// Mitsubishi GX Works2 project: GCP-712ARB(2#)-20040003-220112   PLC: Q03UDV

PROGRAM 01INITI
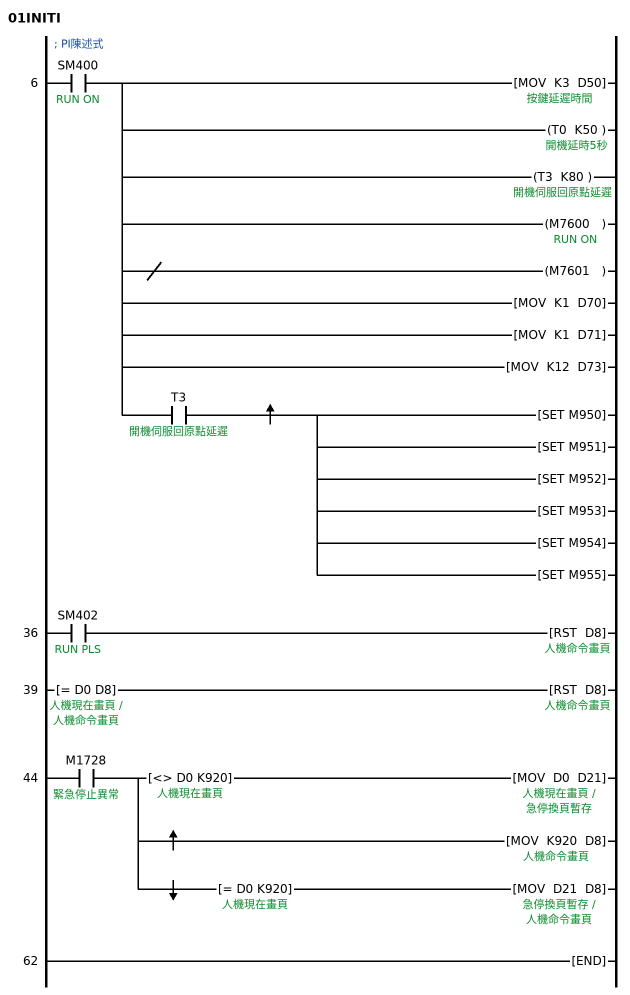
; PI陳述式
6     LD      SM400  ; RUN ON
      MOV     K3 D50  ; 按鍵延遲時間
      OUT     T0 K50  ; 開機延時5秒
      OUT     T3 K80  ; 開機伺服回原點延遲
      OUT     M7600  ; RUN ON
      MPS
      INV
      OUT     M7601
      MPP
      MOV     K1 D70
      MOV     K1 D71
      MOV     K12 D73
      AND     T3  ; 開機伺服回原點延遲
      MEP
      SET     M950
      SET     M951
      SET     M952
      SET     M953
      SET     M954
      SET     M955
36    LD      SM402  ; RUN PLS
      RST     D8  ; 人機命令畫頁
39    LD=     D0 D8  ; 人機現在畫頁 / 人機命令畫頁
      RST     D8  ; 人機命令畫頁
44    LD      M1728  ; 緊急停止異常
      MPS
      AND<>   D0 K920  ; 人機現在畫頁
      MOV     D0 D21  ; 急停換頁暫存
      MRD
      MEP
      MOV     K920 D8
      MPP
      MEF
      AND=    D0 K920  ; 人機現在畫頁
      MOV     D21 D8
62    END
END_PROGRAM

PROGRAM 02FUNC
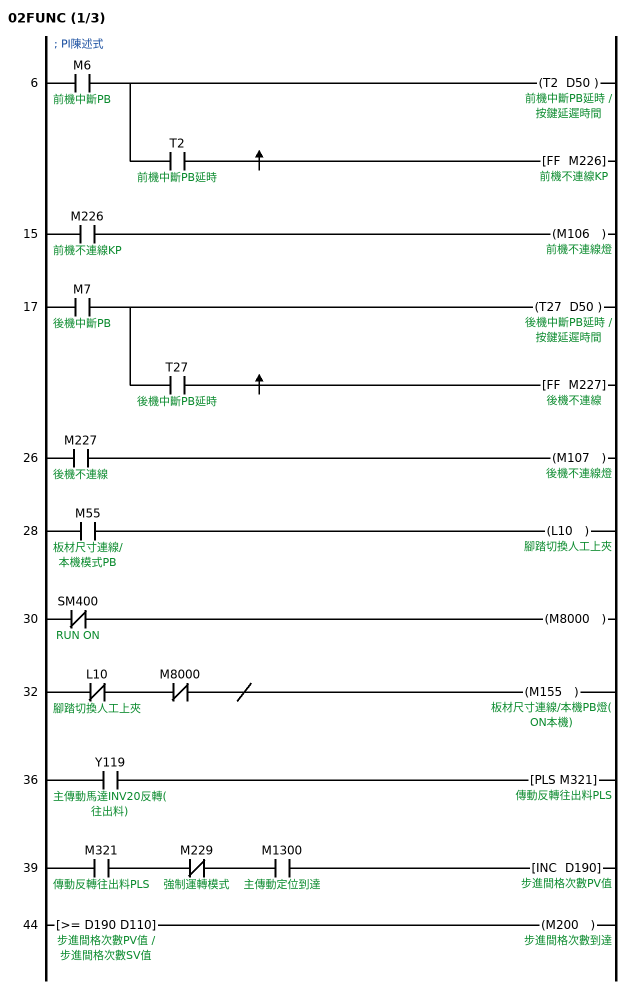
; PI陳述式
6     LD      M6  ; 前機中斷PB
      OUT     T2 D50  ; 前機中斷PB延時 / 按鍵延遲時間
      AND     T2  ; 前機中斷PB延時
      MEP
      FF      M226  ; 前機不連線KP
15    LD      M226  ; 前機不連線KP
      OUT     M106  ; 前機不連線燈
17    LD      M7  ; 後機中斷PB
      OUT     T27 D50  ; 後機中斷PB延時 / 按鍵延遲時間
      AND     T27  ; 後機中斷PB延時
      MEP
      FF      M227  ; 後機不連線
26    LD      M227  ; 後機不連線
      OUT     M107  ; 後機不連線燈
28    LD      M55  ; 板材尺寸連線/本機模式PB
      OUT     L10  ; 腳踏切換人工上夾
30    LDI     SM400  ; RUN ON
      OUT     M8000
32    LDI     L10  ; 腳踏切換人工上夾
      ANI     M8000
      INV
      OUT     M155  ; 板材尺寸連線/本機PB燈(ON本機)
36    LD      Y119  ; 主傳動馬達INV20反轉(往出料)
      PLS     M321  ; 傳動反轉往出料PLS
39    LD      M321  ; 傳動反轉往出料PLS
      ANI     M229  ; 強制運轉模式
      AND     M1300  ; 主傳動定位到達
      INC     D190  ; 步進間格次數PV值
44    LD>=    D190 D110  ; 步進間格次數PV值 / 步進間格次數SV值
      OUT     M200  ; 步進間格次數到達
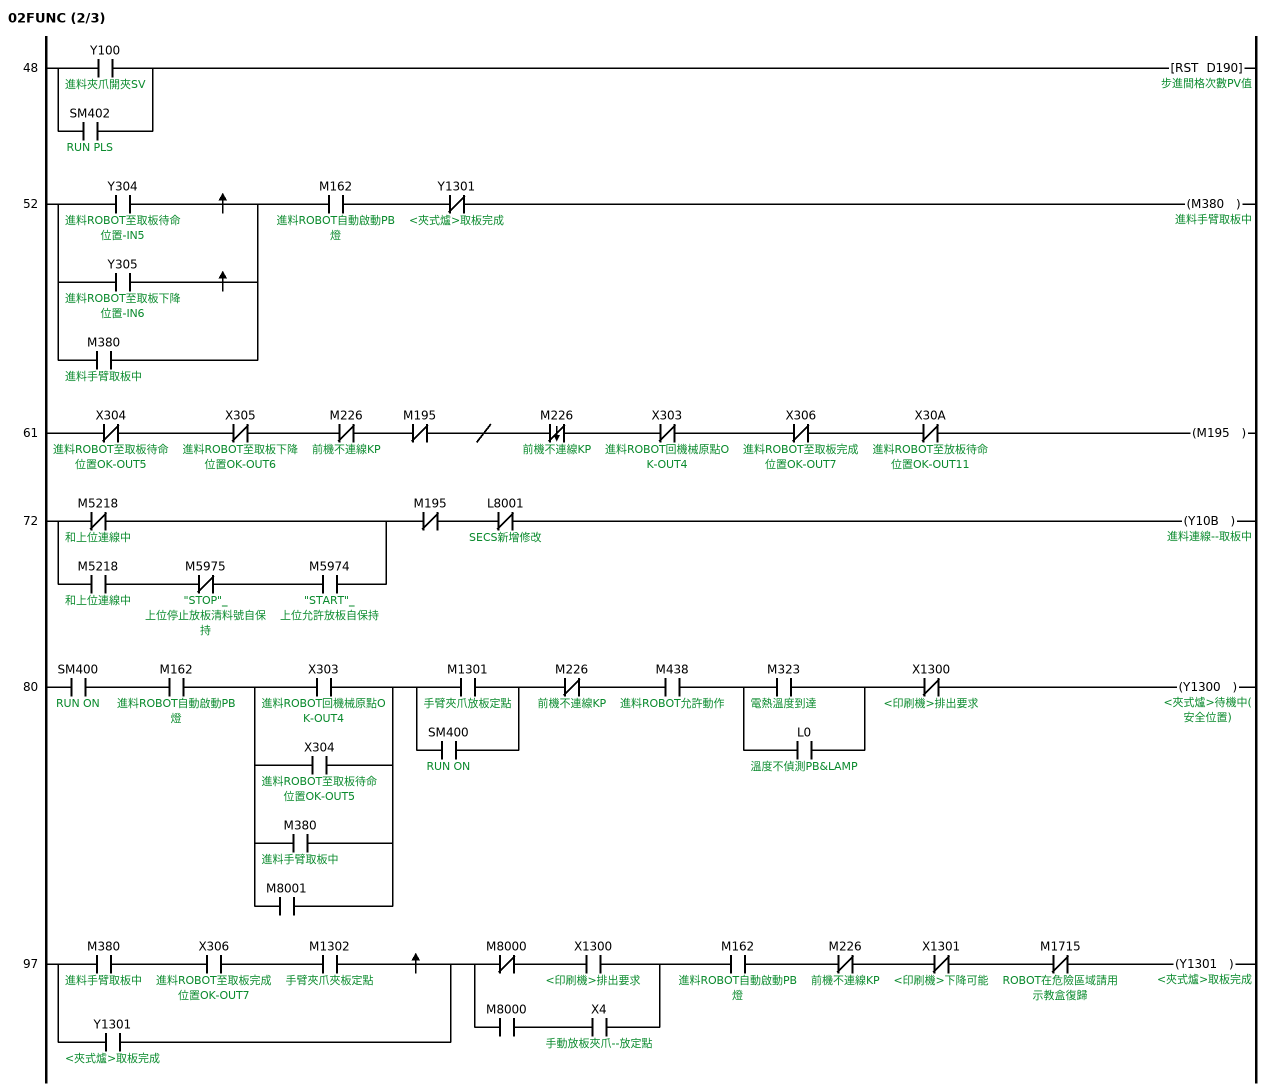
48    LD      Y100  ; 進料夾爪開夾SV
      OR      SM402  ; RUN PLS
      RST     D190  ; 步進間格次數PV值
52    LD      Y304  ; 進料ROBOT至取板待命位置-IN5
      MEP
      LD      Y305  ; 進料ROBOT至取板下降位置-IN6
      MEP
      ORB
      OR      M380  ; 進料手臂取板中
      AND     M162  ; 進料ROBOT自動啟動PB燈
      ANI     Y1301  ; <夾式爐>取板完成
      OUT     M380  ; 進料手臂取板中
61    LDI     X304  ; 進料ROBOT至取板待命位置OK-OUT5
      ANI     X305  ; 進料ROBOT至取板下降位置OK-OUT6
      ANI     M226  ; 前機不連線KP
      ANI     M195
      INV
      ANDFI   M226  ; 前機不連線KP
      ANI     X303  ; 進料ROBOT回機械原點OK-OUT4
      ANI     X306  ; 進料ROBOT至取板完成位置OK-OUT7
      ANI     X30A  ; 進料ROBOT至放板待命位置OK-OUT11
      OUT     M195
72    LDI     M5218  ; 和上位連線中
      LD      M5218  ; 和上位連線中
      ANI     M5975  ; "STOP"_ 上位停止放板清料號自保持
      AND     M5974  ; "START"_上位允許放板自保持
      ORB
      ANI     M195
      ANI     L8001  ; SECS新增修改
      OUT     Y10B  ; 進料連線--取板中
80    LD      SM400  ; RUN ON
      AND     M162  ; 進料ROBOT自動啟動PB燈
      LD      X303  ; 進料ROBOT回機械原點OK-OUT4
      OR      X304  ; 進料ROBOT至取板待命位置OK-OUT5
      OR      M380  ; 進料手臂取板中
      OR      M8001
      ANB
      LD      M1301  ; 手臂夾爪放板定點
      OR      SM400  ; RUN ON
      ANB
      ANI     M226  ; 前機不連線KP
      AND     M438  ; 進料ROBOT允許動作
      LD      M323  ; 電熱溫度到達
      OR      L0  ; 溫度不偵測PB&LAMP
      ANB
      ANI     X1300  ; <印刷機>排出要求
      OUT     Y1300  ; <夾式爐>待機中(安全位置)
97    LD      M380  ; 進料手臂取板中
      AND     X306  ; 進料ROBOT至取板完成位置OK-OUT7
      AND     M1302  ; 手臂夾爪夾板定點
      MEP
      OR      Y1301  ; <夾式爐>取板完成
      LDI     M8000
      AND     X1300  ; <印刷機>排出要求
      LD      M8000
      AND     X4  ; 手動放板夾爪--放定點
      ORB
      ANB
      AND     M162  ; 進料ROBOT自動啟動PB燈
      ANI     M226  ; 前機不連線KP
      ANI     X1301  ; <印刷機>下降可能
      ANI     M1715  ; ROBOT在危險區域請用示教盒復歸
      OUT     Y1301  ; <夾式爐>取板完成
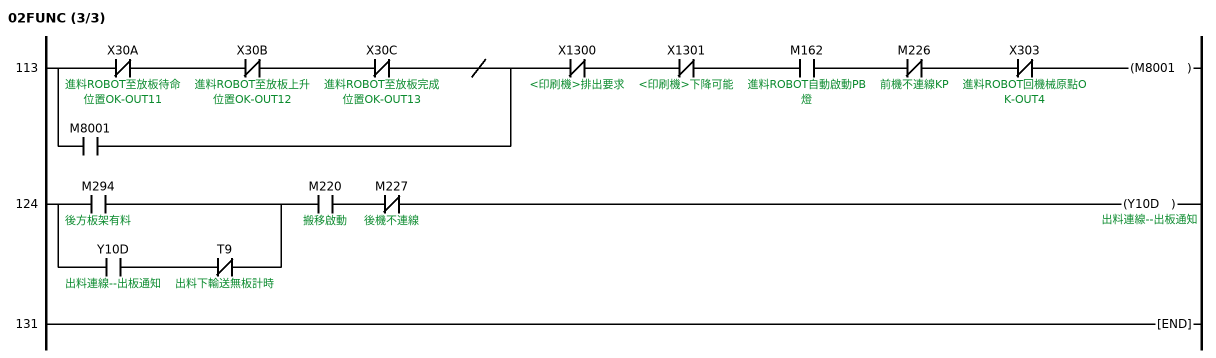
113   LDI     X30A  ; 進料ROBOT至放板待命位置OK-OUT11
      ANI     X30B  ; 進料ROBOT至放板上升位置OK-OUT12
      ANI     X30C  ; 進料ROBOT至放板完成位置OK-OUT13
      INV
      OR      M8001
      ANI     X1300  ; <印刷機>排出要求
      ANI     X1301  ; <印刷機>下降可能
      AND     M162  ; 進料ROBOT自動啟動PB燈
      ANI     M226  ; 前機不連線KP
      ANI     X303  ; 進料ROBOT回機械原點OK-OUT4
      OUT     M8001
124   LD      M294  ; 後方板架有料
      LD      Y10D  ; 出料連線--出板通知
      ANI     T9  ; 出料下輸送無板計時
      ORB
      AND     M220  ; 搬移啟動
      ANI     M227  ; 後機不連線
      OUT     Y10D  ; 出料連線--出板通知
131   END
END_PROGRAM

PROGRAM 03ORIGIN
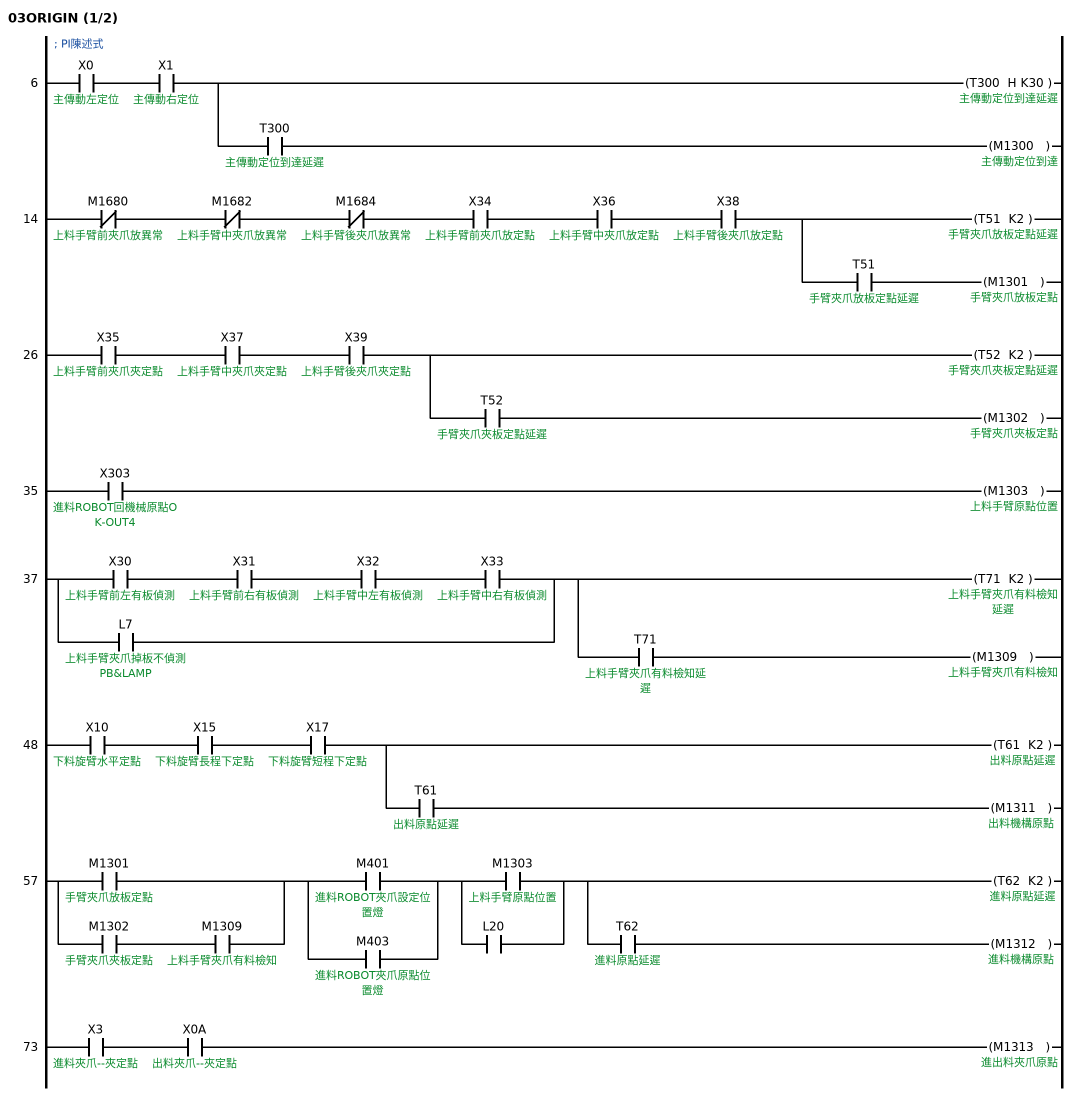
; PI陳述式
6     LD      X0  ; 主傳動左定位
      AND     X1  ; 主傳動右定位
      OUTH    T300 K30  ; 主傳動定位到達延遲
      AND     T300  ; 主傳動定位到達延遲
      OUT     M1300  ; 主傳動定位到達
14    LDI     M1680  ; 上料手臂前夾爪放異常
      ANI     M1682  ; 上料手臂中夾爪放異常
      ANI     M1684  ; 上料手臂後夾爪放異常
      AND     X34  ; 上料手臂前夾爪放定點
      AND     X36  ; 上料手臂中夾爪放定點
      AND     X38  ; 上料手臂後夾爪放定點
      OUT     T51 K2  ; 手臂夾爪放板定點延遲
      AND     T51  ; 手臂夾爪放板定點延遲
      OUT     M1301  ; 手臂夾爪放板定點
26    LD      X35  ; 上料手臂前夾爪夾定點
      AND     X37  ; 上料手臂中夾爪夾定點
      AND     X39  ; 上料手臂後夾爪夾定點
      OUT     T52 K2  ; 手臂夾爪夾板定點延遲
      AND     T52  ; 手臂夾爪夾板定點延遲
      OUT     M1302  ; 手臂夾爪夾板定點
35    LD      X303  ; 進料ROBOT回機械原點OK-OUT4
      OUT     M1303  ; 上料手臂原點位置
37    LD      X30  ; 上料手臂前左有板偵測
      AND     X31  ; 上料手臂前右有板偵測
      AND     X32  ; 上料手臂中左有板偵測
      AND     X33  ; 上料手臂中右有板偵測
      OR      L7  ; 上料手臂夾爪掉板不偵測PB&LAMP
      OUT     T71 K2  ; 上料手臂夾爪有料檢知延遲
      AND     T71  ; 上料手臂夾爪有料檢知延遲
      OUT     M1309  ; 上料手臂夾爪有料檢知
48    LD      X10  ; 下料旋臂水平定點
      AND     X15  ; 下料旋臂長程下定點
      AND     X17  ; 下料旋臂短程下定點
      OUT     T61 K2  ; 出料原點延遲
      AND     T61  ; 出料原點延遲
      OUT     M1311  ; 出料機構原點
57    LD      M1301  ; 手臂夾爪放板定點
      LD      M1302  ; 手臂夾爪夾板定點
      AND     M1309  ; 上料手臂夾爪有料檢知
      ORB
      LD      M401  ; 進料ROBOT夾爪設定位置燈
      OR      M403  ; 進料ROBOT夾爪原點位置燈
      ANB
      LD      M1303  ; 上料手臂原點位置
      OR      L20
      ANB
      OUT     T62 K2  ; 進料原點延遲
      AND     T62  ; 進料原點延遲
      OUT     M1312  ; 進料機構原點
73    LD      X3  ; 進料夾爪--夾定點
      AND     X0A  ; 出料夾爪--夾定點
      OUT     M1313  ; 進出料夾爪原點
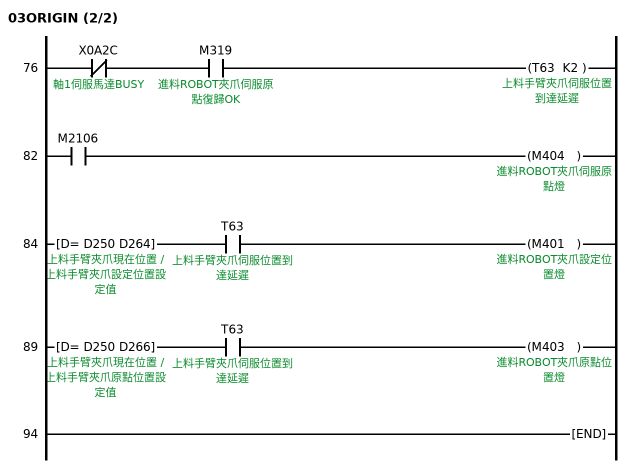
76    LDI     X0A2C  ; 軸1伺服馬達BUSY
      AND     M319  ; 進料ROBOT夾爪伺服原點復歸OK
      OUT     T63 K2  ; 上料手臂夾爪伺服位置到達延遲
82    LD      M2106
      OUT     M404  ; 進料ROBOT夾爪伺服原點燈
84    LDD=    D250 D264  ; 上料手臂夾爪現在位置 / 上料手臂夾爪設定位置設定值
      AND     T63  ; 上料手臂夾爪伺服位置到達延遲
      OUT     M401  ; 進料ROBOT夾爪設定位置燈
89    LDD=    D250 D266  ; 上料手臂夾爪現在位置 / 上料手臂夾爪原點位置設定值
      AND     T63  ; 上料手臂夾爪伺服位置到達延遲
      OUT     M403  ; 進料ROBOT夾爪原點位置燈
94    END
END_PROGRAM

PROGRAM 04LOAD
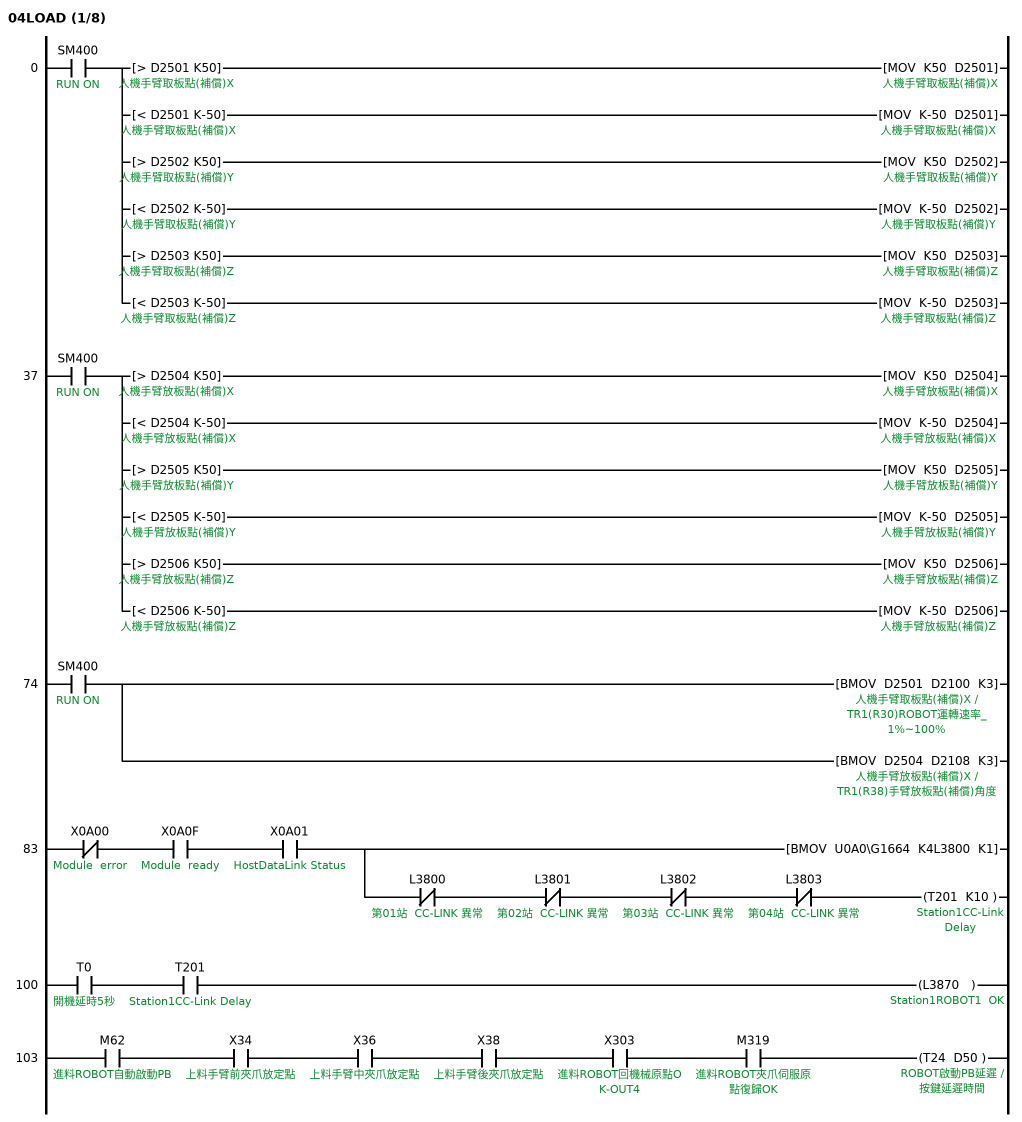
0     LD      SM400  ; RUN ON
      MPS
      AND>    D2501 K50  ; 人機手臂取板點(補償)X
      MOV     K50 D2501
      MRD
      AND<    D2501 K-50  ; 人機手臂取板點(補償)X
      MOV     K-50 D2501
      MRD
      AND>    D2502 K50  ; 人機手臂取板點(補償)Y
      MOV     K50 D2502
      MRD
      AND<    D2502 K-50  ; 人機手臂取板點(補償)Y
      MOV     K-50 D2502
      MRD
      AND>    D2503 K50  ; 人機手臂取板點(補償)Z
      MOV     K50 D2503
      MPP
      AND<    D2503 K-50  ; 人機手臂取板點(補償)Z
      MOV     K-50 D2503
37    LD      SM400  ; RUN ON
      MPS
      AND>    D2504 K50  ; 人機手臂放板點(補償)X
      MOV     K50 D2504
      MRD
      AND<    D2504 K-50  ; 人機手臂放板點(補償)X
      MOV     K-50 D2504
      MRD
      AND>    D2505 K50  ; 人機手臂放板點(補償)Y
      MOV     K50 D2505
      MRD
      AND<    D2505 K-50  ; 人機手臂放板點(補償)Y
      MOV     K-50 D2505
      MRD
      AND>    D2506 K50  ; 人機手臂放板點(補償)Z
      MOV     K50 D2506
      MPP
      AND<    D2506 K-50  ; 人機手臂放板點(補償)Z
      MOV     K-50 D2506
74    LD      SM400  ; RUN ON
      BMOV    D2501 D2100 K3  ; TR1(R30)ROBOT運轉速率_1%~100%
      BMOV    D2504 D2108 K3  ; TR1(R38)手臂放板點(補償)角度
83    LDI     X0A00  ; Module  error
      AND     X0A0F  ; Module  ready
      AND     X0A01  ; HostDataLink Status
      BMOV    U0A0\G1664 K4L3800 K1  ; 第01站  CC-LINK 異常
      ANI     L3800  ; 第01站  CC-LINK 異常
      ANI     L3801  ; 第02站  CC-LINK 異常
      ANI     L3802  ; 第03站  CC-LINK 異常
      ANI     L3803  ; 第04站  CC-LINK 異常
      OUT     T201 K10  ; Station1CC-Link Delay
100   LD      T0  ; 開機延時5秒
      AND     T201  ; Station1CC-Link Delay
      OUT     L3870  ; Station1ROBOT1  OK
103   LD      M62  ; 進料ROBOT自動啟動PB
      AND     X34  ; 上料手臂前夾爪放定點
      AND     X36  ; 上料手臂中夾爪放定點
      AND     X38  ; 上料手臂後夾爪放定點
      AND     X303  ; 進料ROBOT回機械原點OK-OUT4
      AND     M319  ; 進料ROBOT夾爪伺服原點復歸OK
      OUT     T24 D50  ; ROBOT啟動PB延遲 / 按鍵延遲時間
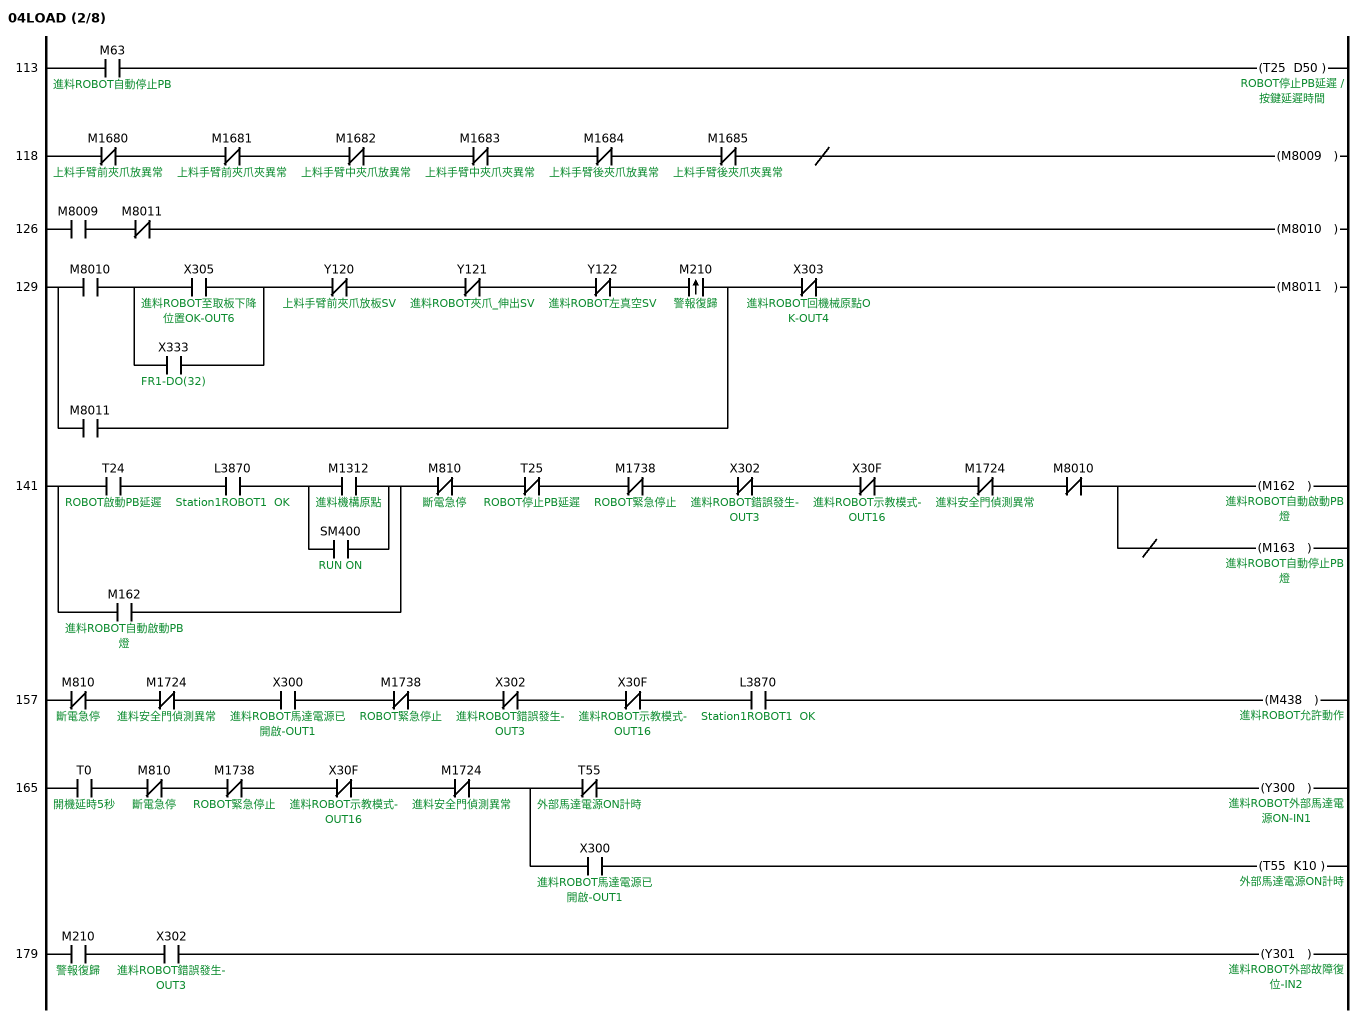
113   LD      M63  ; 進料ROBOT自動停止PB
      OUT     T25 D50  ; ROBOT停止PB延遲 / 按鍵延遲時間
118   LDI     M1680  ; 上料手臂前夾爪放異常
      ANI     M1681  ; 上料手臂前夾爪夾異常
      ANI     M1682  ; 上料手臂中夾爪放異常
      ANI     M1683  ; 上料手臂中夾爪夾異常
      ANI     M1684  ; 上料手臂後夾爪放異常
      ANI     M1685  ; 上料手臂後夾爪夾異常
      INV
      OUT     M8009
126   LD      M8009
      ANI     M8011
      OUT     M8010
129   LD      M8010
      LD      X305  ; 進料ROBOT至取板下降位置OK-OUT6
      OR      X333  ; FR1-DO(32)
      ANB
      ANI     Y120  ; 上料手臂前夾爪放板SV
      ANI     Y121  ; 進料ROBOT夾爪_伸出SV
      ANI     Y122  ; 進料ROBOT左真空SV
      ANDP    M210  ; 警報復歸
      OR      M8011
      ANI     X303  ; 進料ROBOT回機械原點OK-OUT4
      OUT     M8011
141   LD      T24  ; ROBOT啟動PB延遲
      AND     L3870  ; Station1ROBOT1  OK
      LD      M1312  ; 進料機構原點
      OR      SM400  ; RUN ON
      ANB
      OR      M162  ; 進料ROBOT自動啟動PB燈
      ANI     M810  ; 斷電急停
      ANI     T25  ; ROBOT停止PB延遲
      ANI     M1738  ; ROBOT緊急停止
      ANI     X302  ; 進料ROBOT錯誤發生-OUT3
      ANI     X30F  ; 進料ROBOT示教模式-OUT16
      ANI     M1724  ; 進料安全門偵測異常
      ANI     M8010
      OUT     M162  ; 進料ROBOT自動啟動PB燈
      INV
      OUT     M163  ; 進料ROBOT自動停止PB燈
157   LDI     M810  ; 斷電急停
      ANI     M1724  ; 進料安全門偵測異常
      AND     X300  ; 進料ROBOT馬達電源已開啟-OUT1
      ANI     M1738  ; ROBOT緊急停止
      ANI     X302  ; 進料ROBOT錯誤發生-OUT3
      ANI     X30F  ; 進料ROBOT示教模式-OUT16
      AND     L3870  ; Station1ROBOT1  OK
      OUT     M438  ; 進料ROBOT允許動作
165   LD      T0  ; 開機延時5秒
      ANI     M810  ; 斷電急停
      ANI     M1738  ; ROBOT緊急停止
      ANI     X30F  ; 進料ROBOT示教模式-OUT16
      ANI     M1724  ; 進料安全門偵測異常
      MPS
      ANI     T55  ; 外部馬達電源ON計時
      OUT     Y300  ; 進料ROBOT外部馬達電源ON-IN1
      MPP
      AND     X300  ; 進料ROBOT馬達電源已開啟-OUT1
      OUT     T55 K10  ; 外部馬達電源ON計時
179   LD      M210  ; 警報復歸
      AND     X302  ; 進料ROBOT錯誤發生-OUT3
      OUT     Y301  ; 進料ROBOT外部故障復位-IN2
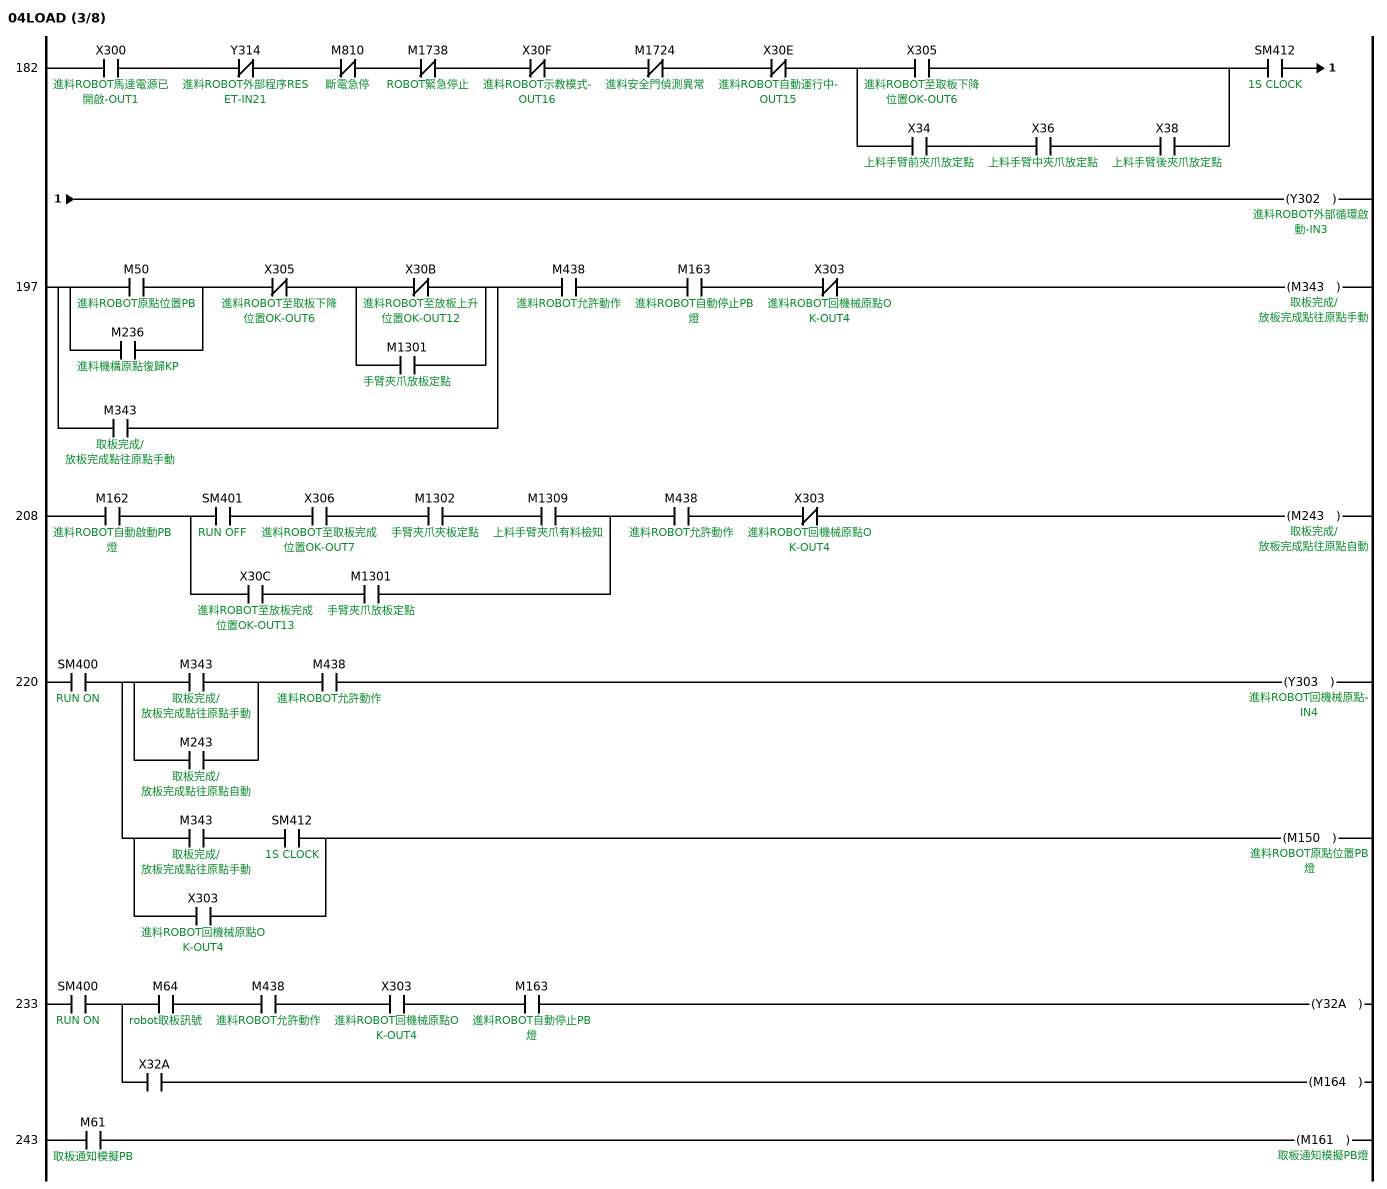
182   LD      X300  ; 進料ROBOT馬達電源已開啟-OUT1
      ANI     Y314  ; 進料ROBOT外部程序RESET-IN21
      ANI     M810  ; 斷電急停
      ANI     M1738  ; ROBOT緊急停止
      ANI     X30F  ; 進料ROBOT示教模式-OUT16
      ANI     M1724  ; 進料安全門偵測異常
      ANI     X30E  ; 進料ROBOT自動運行中-OUT15
      LD      X305  ; 進料ROBOT至取板下降位置OK-OUT6
      LD      X34  ; 上料手臂前夾爪放定點
      AND     X36  ; 上料手臂中夾爪放定點
      AND     X38  ; 上料手臂後夾爪放定點
      ORB
      ANB
      AND     SM412  ; 1S CLOCK
      OUT     Y302  ; 進料ROBOT外部循環啟動-IN3
197   LD      M50  ; 進料ROBOT原點位置PB
      OR      M236  ; 進料機構原點復歸KP
      ANI     X305  ; 進料ROBOT至取板下降位置OK-OUT6
      LDI     X30B  ; 進料ROBOT至放板上升位置OK-OUT12
      OR      M1301  ; 手臂夾爪放板定點
      ANB
      OR      M343  ; 取板完成/放板完成點往原點手動
      AND     M438  ; 進料ROBOT允許動作
      AND     M163  ; 進料ROBOT自動停止PB燈
      ANI     X303  ; 進料ROBOT回機械原點OK-OUT4
      OUT     M343  ; 取板完成/放板完成點往原點手動
208   LD      M162  ; 進料ROBOT自動啟動PB燈
      LD      SM401  ; RUN OFF
      AND     X306  ; 進料ROBOT至取板完成位置OK-OUT7
      AND     M1302  ; 手臂夾爪夾板定點
      AND     M1309  ; 上料手臂夾爪有料檢知
      LD      X30C  ; 進料ROBOT至放板完成位置OK-OUT13
      AND     M1301  ; 手臂夾爪放板定點
      ORB
      ANB
      AND     M438  ; 進料ROBOT允許動作
      ANI     X303  ; 進料ROBOT回機械原點OK-OUT4
      OUT     M243  ; 取板完成/放板完成點往原點自動
220   LD      SM400  ; RUN ON
      MPS
      LD      M343  ; 取板完成/放板完成點往原點手動
      OR      M243  ; 取板完成/放板完成點往原點自動
      ANB
      AND     M438  ; 進料ROBOT允許動作
      OUT     Y303  ; 進料ROBOT回機械原點-IN4
      MPP
      LD      M343  ; 取板完成/放板完成點往原點手動
      AND     SM412  ; 1S CLOCK
      OR      X303  ; 進料ROBOT回機械原點OK-OUT4
      ANB
      OUT     M150  ; 進料ROBOT原點位置PB燈
233   LD      SM400  ; RUN ON
      MPS
      AND     M64  ; robot取板訊號
      AND     M438  ; 進料ROBOT允許動作
      AND     X303  ; 進料ROBOT回機械原點OK-OUT4
      AND     M163  ; 進料ROBOT自動停止PB燈
      OUT     Y32A
      MPP
      AND     X32A
      OUT     M164
243   LD      M61  ; 取板通知模擬PB
      OUT     M161  ; 取板通知模擬PB燈
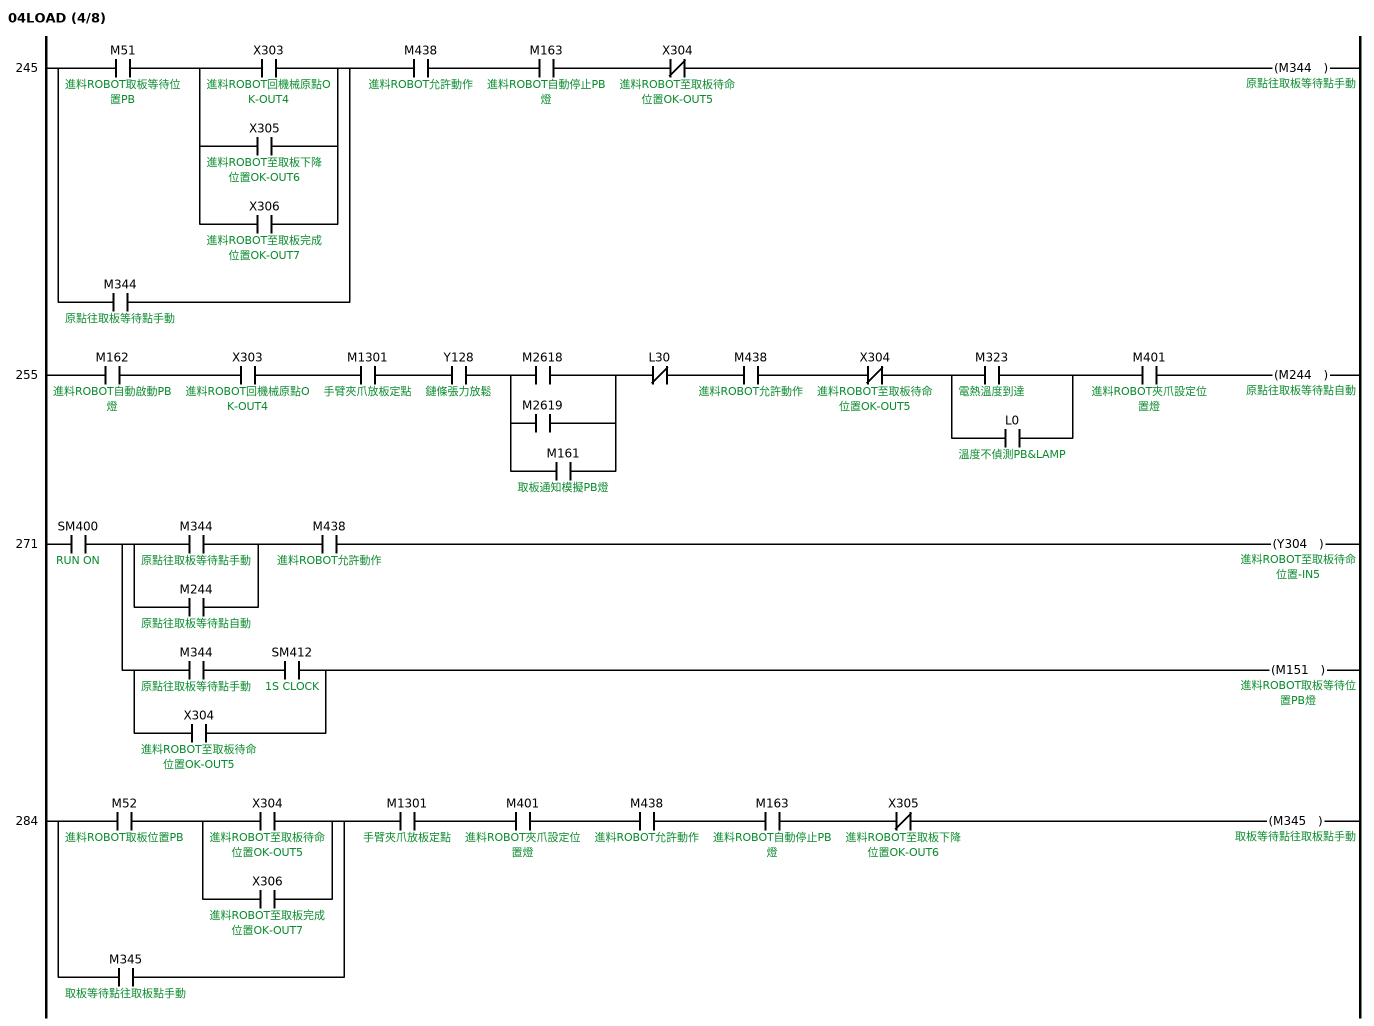
245   LD      M51  ; 進料ROBOT取板等待位置PB
      LD      X303  ; 進料ROBOT回機械原點OK-OUT4
      OR      X305  ; 進料ROBOT至取板下降位置OK-OUT6
      OR      X306  ; 進料ROBOT至取板完成位置OK-OUT7
      ANB
      OR      M344  ; 原點往取板等待點手動
      AND     M438  ; 進料ROBOT允許動作
      AND     M163  ; 進料ROBOT自動停止PB燈
      ANI     X304  ; 進料ROBOT至取板待命位置OK-OUT5
      OUT     M344  ; 原點往取板等待點手動
255   LD      M162  ; 進料ROBOT自動啟動PB燈
      AND     X303  ; 進料ROBOT回機械原點OK-OUT4
      AND     M1301  ; 手臂夾爪放板定點
      AND     Y128  ; 鏈條張力放鬆
      LD      M2618
      OR      M2619
      OR      M161  ; 取板通知模擬PB燈
      ANB
      ANI     L30
      AND     M438  ; 進料ROBOT允許動作
      ANI     X304  ; 進料ROBOT至取板待命位置OK-OUT5
      LD      M323  ; 電熱溫度到達
      OR      L0  ; 溫度不偵測PB&LAMP
      ANB
      AND     M401  ; 進料ROBOT夾爪設定位置燈
      OUT     M244  ; 原點往取板等待點自動
271   LD      SM400  ; RUN ON
      MPS
      LD      M344  ; 原點往取板等待點手動
      OR      M244  ; 原點往取板等待點自動
      ANB
      AND     M438  ; 進料ROBOT允許動作
      OUT     Y304  ; 進料ROBOT至取板待命位置-IN5
      MPP
      LD      M344  ; 原點往取板等待點手動
      AND     SM412  ; 1S CLOCK
      OR      X304  ; 進料ROBOT至取板待命位置OK-OUT5
      ANB
      OUT     M151  ; 進料ROBOT取板等待位置PB燈
284   LD      M52  ; 進料ROBOT取板位置PB
      LD      X304  ; 進料ROBOT至取板待命位置OK-OUT5
      OR      X306  ; 進料ROBOT至取板完成位置OK-OUT7
      ANB
      OR      M345  ; 取板等待點往取板點手動
      AND     M1301  ; 手臂夾爪放板定點
      AND     M401  ; 進料ROBOT夾爪設定位置燈
      AND     M438  ; 進料ROBOT允許動作
      AND     M163  ; 進料ROBOT自動停止PB燈
      ANI     X305  ; 進料ROBOT至取板下降位置OK-OUT6
      OUT     M345  ; 取板等待點往取板點手動
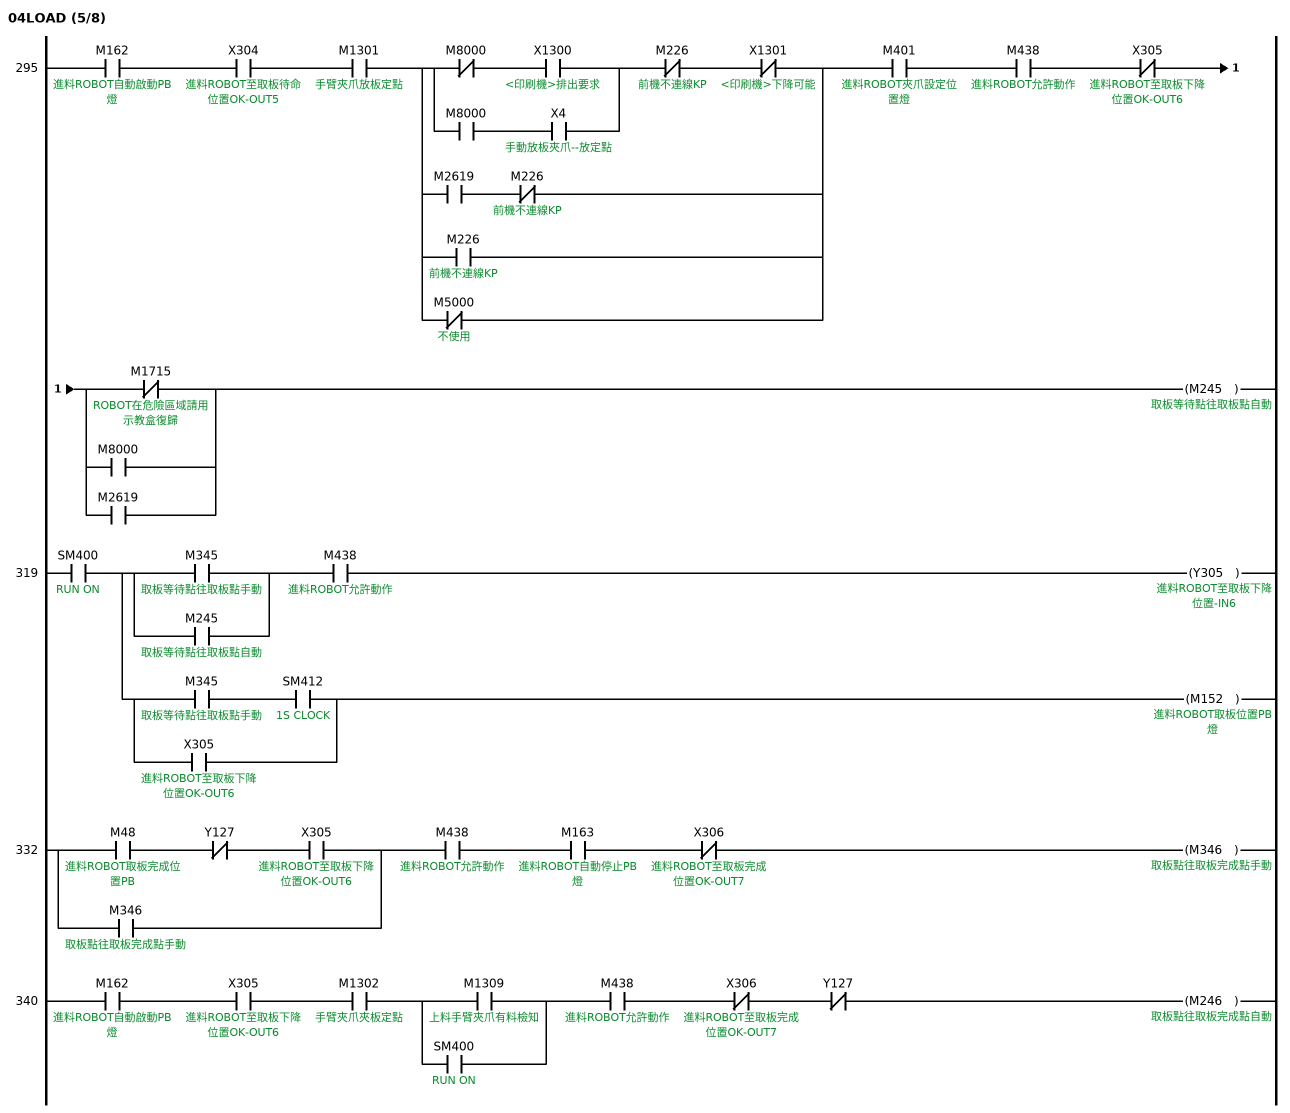
295   LD      M162  ; 進料ROBOT自動啟動PB燈
      AND     X304  ; 進料ROBOT至取板待命位置OK-OUT5
      AND     M1301  ; 手臂夾爪放板定點
      LDI     M8000
      AND     X1300  ; <印刷機>排出要求
      LD      M8000
      AND     X4  ; 手動放板夾爪--放定點
      ORB
      ANI     M226  ; 前機不連線KP
      ANI     X1301  ; <印刷機>下降可能
      LD      M2619
      ANI     M226  ; 前機不連線KP
      ORB
      OR      M226  ; 前機不連線KP
      ORI     M5000  ; 不使用
      ANB
      AND     M401  ; 進料ROBOT夾爪設定位置燈
      AND     M438  ; 進料ROBOT允許動作
      ANI     X305  ; 進料ROBOT至取板下降位置OK-OUT6
      LDI     M1715  ; ROBOT在危險區域請用示教盒復歸
      OR      M8000
      OR      M2619
      ANB
      OUT     M245  ; 取板等待點往取板點自動
319   LD      SM400  ; RUN ON
      MPS
      LD      M345  ; 取板等待點往取板點手動
      OR      M245  ; 取板等待點往取板點自動
      ANB
      AND     M438  ; 進料ROBOT允許動作
      OUT     Y305  ; 進料ROBOT至取板下降位置-IN6
      MPP
      LD      M345  ; 取板等待點往取板點手動
      AND     SM412  ; 1S CLOCK
      OR      X305  ; 進料ROBOT至取板下降位置OK-OUT6
      ANB
      OUT     M152  ; 進料ROBOT取板位置PB燈
332   LD      M48  ; 進料ROBOT取板完成位置PB
      ANI     Y127
      AND     X305  ; 進料ROBOT至取板下降位置OK-OUT6
      OR      M346  ; 取板點往取板完成點手動
      AND     M438  ; 進料ROBOT允許動作
      AND     M163  ; 進料ROBOT自動停止PB燈
      ANI     X306  ; 進料ROBOT至取板完成位置OK-OUT7
      OUT     M346  ; 取板點往取板完成點手動
340   LD      M162  ; 進料ROBOT自動啟動PB燈
      AND     X305  ; 進料ROBOT至取板下降位置OK-OUT6
      AND     M1302  ; 手臂夾爪夾板定點
      LD      M1309  ; 上料手臂夾爪有料檢知
      OR      SM400  ; RUN ON
      ANB
      AND     M438  ; 進料ROBOT允許動作
      ANI     X306  ; 進料ROBOT至取板完成位置OK-OUT7
      ANI     Y127
      OUT     M246  ; 取板點往取板完成點自動
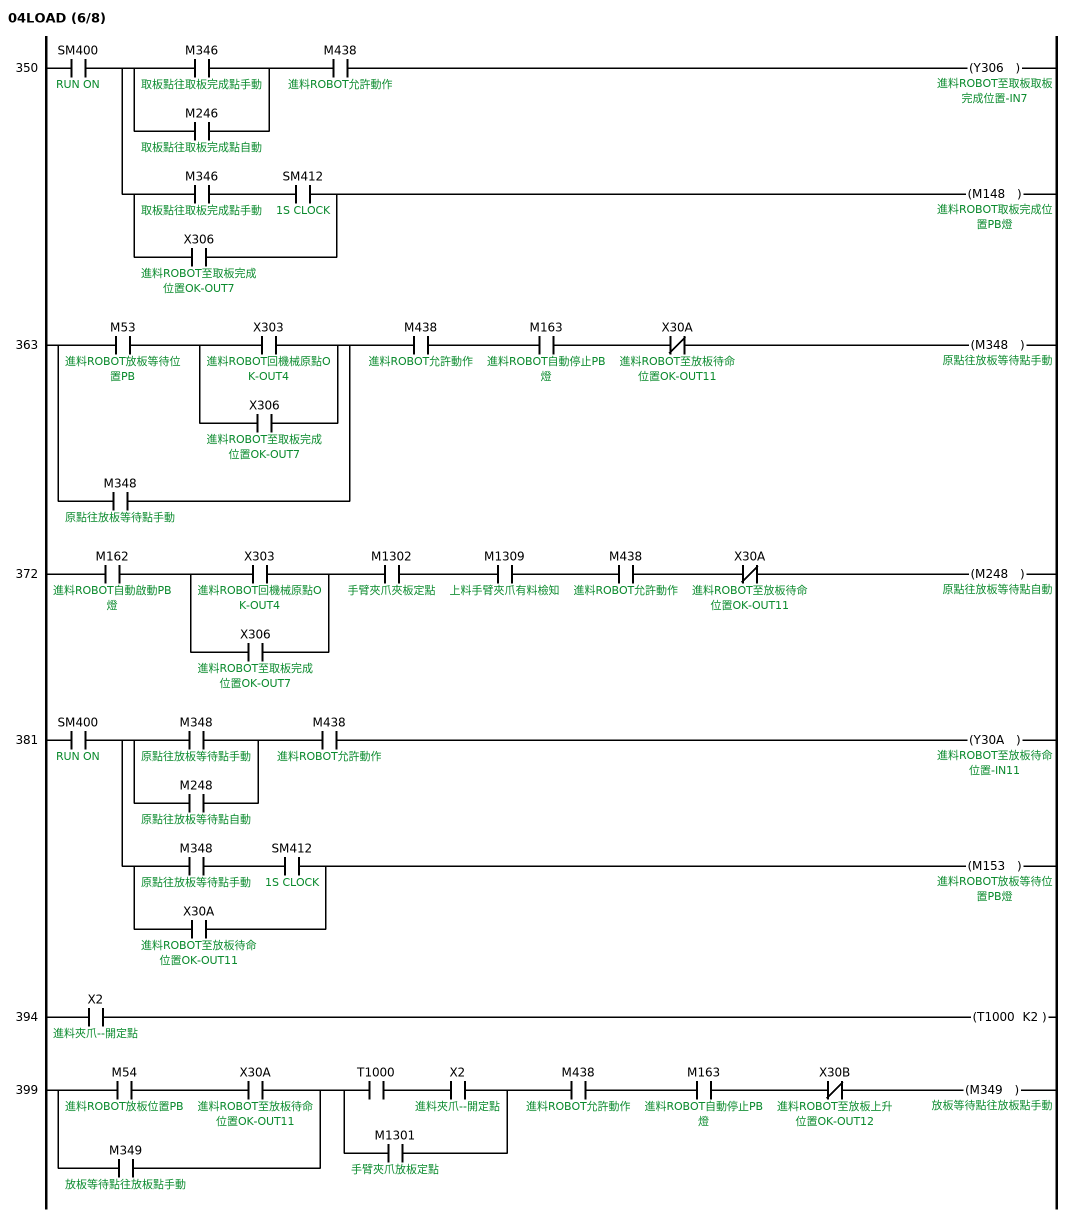
350   LD      SM400  ; RUN ON
      MPS
      LD      M346  ; 取板點往取板完成點手動
      OR      M246  ; 取板點往取板完成點自動
      ANB
      AND     M438  ; 進料ROBOT允許動作
      OUT     Y306  ; 進料ROBOT至取板取板完成位置-IN7
      MPP
      LD      M346  ; 取板點往取板完成點手動
      AND     SM412  ; 1S CLOCK
      OR      X306  ; 進料ROBOT至取板完成位置OK-OUT7
      ANB
      OUT     M148  ; 進料ROBOT取板完成位置PB燈
363   LD      M53  ; 進料ROBOT放板等待位置PB
      LD      X303  ; 進料ROBOT回機械原點OK-OUT4
      OR      X306  ; 進料ROBOT至取板完成位置OK-OUT7
      ANB
      OR      M348  ; 原點往放板等待點手動
      AND     M438  ; 進料ROBOT允許動作
      AND     M163  ; 進料ROBOT自動停止PB燈
      ANI     X30A  ; 進料ROBOT至放板待命位置OK-OUT11
      OUT     M348  ; 原點往放板等待點手動
372   LD      M162  ; 進料ROBOT自動啟動PB燈
      LD      X303  ; 進料ROBOT回機械原點OK-OUT4
      OR      X306  ; 進料ROBOT至取板完成位置OK-OUT7
      ANB
      AND     M1302  ; 手臂夾爪夾板定點
      AND     M1309  ; 上料手臂夾爪有料檢知
      AND     M438  ; 進料ROBOT允許動作
      ANI     X30A  ; 進料ROBOT至放板待命位置OK-OUT11
      OUT     M248  ; 原點往放板等待點自動
381   LD      SM400  ; RUN ON
      MPS
      LD      M348  ; 原點往放板等待點手動
      OR      M248  ; 原點往放板等待點自動
      ANB
      AND     M438  ; 進料ROBOT允許動作
      OUT     Y30A  ; 進料ROBOT至放板待命位置-IN11
      MPP
      LD      M348  ; 原點往放板等待點手動
      AND     SM412  ; 1S CLOCK
      OR      X30A  ; 進料ROBOT至放板待命位置OK-OUT11
      ANB
      OUT     M153  ; 進料ROBOT放板等待位置PB燈
394   LD      X2  ; 進料夾爪--開定點
      OUT     T1000 K2
399   LD      M54  ; 進料ROBOT放板位置PB
      AND     X30A  ; 進料ROBOT至放板待命位置OK-OUT11
      OR      M349  ; 放板等待點往放板點手動
      LD      T1000
      AND     X2  ; 進料夾爪--開定點
      OR      M1301  ; 手臂夾爪放板定點
      ANB
      AND     M438  ; 進料ROBOT允許動作
      AND     M163  ; 進料ROBOT自動停止PB燈
      ANI     X30B  ; 進料ROBOT至放板上升位置OK-OUT12
      OUT     M349  ; 放板等待點往放板點手動
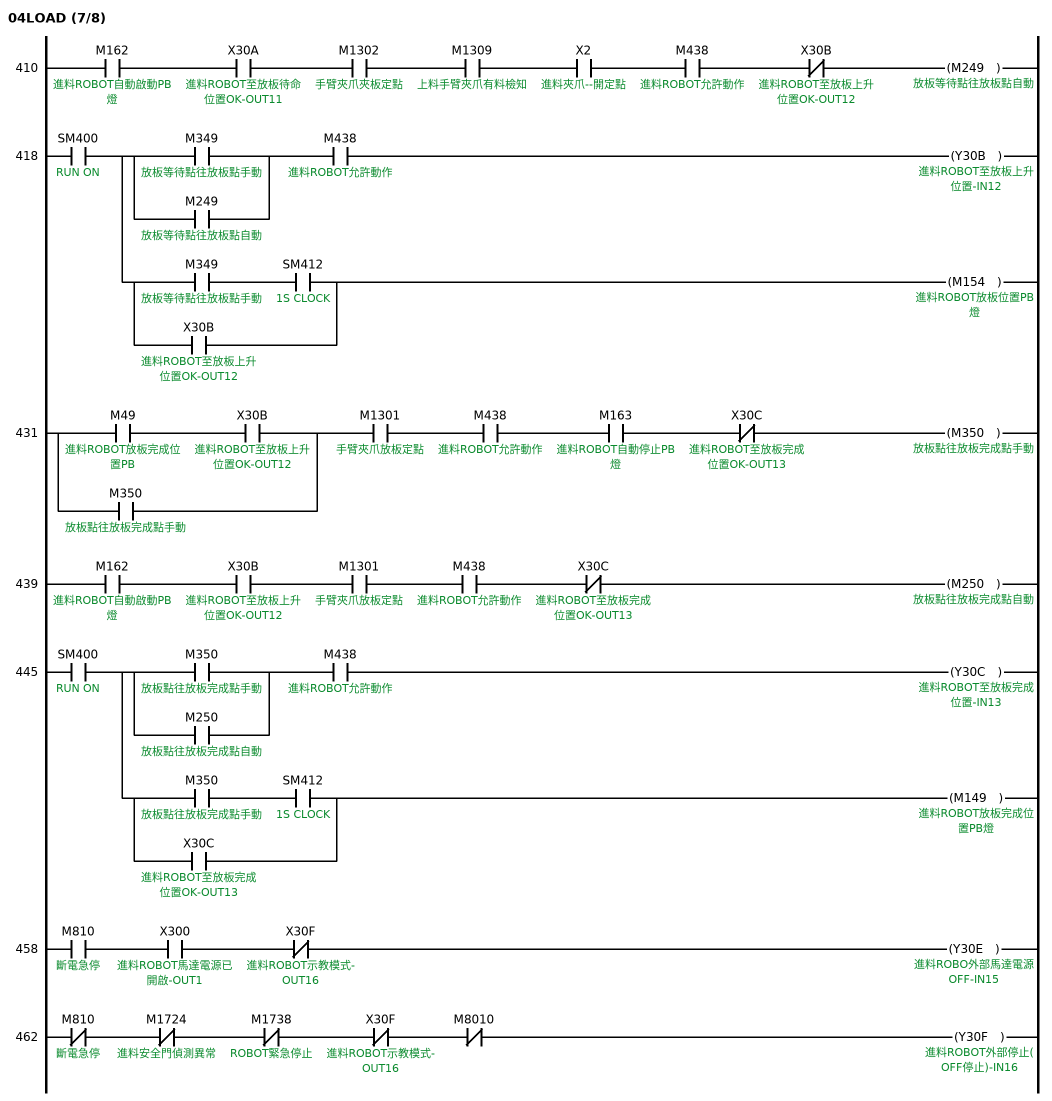
410   LD      M162  ; 進料ROBOT自動啟動PB燈
      AND     X30A  ; 進料ROBOT至放板待命位置OK-OUT11
      AND     M1302  ; 手臂夾爪夾板定點
      AND     M1309  ; 上料手臂夾爪有料檢知
      AND     X2  ; 進料夾爪--開定點
      AND     M438  ; 進料ROBOT允許動作
      ANI     X30B  ; 進料ROBOT至放板上升位置OK-OUT12
      OUT     M249  ; 放板等待點往放板點自動
418   LD      SM400  ; RUN ON
      MPS
      LD      M349  ; 放板等待點往放板點手動
      OR      M249  ; 放板等待點往放板點自動
      ANB
      AND     M438  ; 進料ROBOT允許動作
      OUT     Y30B  ; 進料ROBOT至放板上升位置-IN12
      MPP
      LD      M349  ; 放板等待點往放板點手動
      AND     SM412  ; 1S CLOCK
      OR      X30B  ; 進料ROBOT至放板上升位置OK-OUT12
      ANB
      OUT     M154  ; 進料ROBOT放板位置PB燈
431   LD      M49  ; 進料ROBOT放板完成位置PB
      AND     X30B  ; 進料ROBOT至放板上升位置OK-OUT12
      OR      M350  ; 放板點往放板完成點手動
      AND     M1301  ; 手臂夾爪放板定點
      AND     M438  ; 進料ROBOT允許動作
      AND     M163  ; 進料ROBOT自動停止PB燈
      ANI     X30C  ; 進料ROBOT至放板完成位置OK-OUT13
      OUT     M350  ; 放板點往放板完成點手動
439   LD      M162  ; 進料ROBOT自動啟動PB燈
      AND     X30B  ; 進料ROBOT至放板上升位置OK-OUT12
      AND     M1301  ; 手臂夾爪放板定點
      AND     M438  ; 進料ROBOT允許動作
      ANI     X30C  ; 進料ROBOT至放板完成位置OK-OUT13
      OUT     M250  ; 放板點往放板完成點自動
445   LD      SM400  ; RUN ON
      MPS
      LD      M350  ; 放板點往放板完成點手動
      OR      M250  ; 放板點往放板完成點自動
      ANB
      AND     M438  ; 進料ROBOT允許動作
      OUT     Y30C  ; 進料ROBOT至放板完成位置-IN13
      MPP
      LD      M350  ; 放板點往放板完成點手動
      AND     SM412  ; 1S CLOCK
      OR      X30C  ; 進料ROBOT至放板完成位置OK-OUT13
      ANB
      OUT     M149  ; 進料ROBOT放板完成位置PB燈
458   LD      M810  ; 斷電急停
      AND     X300  ; 進料ROBOT馬達電源已開啟-OUT1
      ANI     X30F  ; 進料ROBOT示教模式-OUT16
      OUT     Y30E  ; 進料ROBO外部馬達電源OFF-IN15
462   LDI     M810  ; 斷電急停
      ANI     M1724  ; 進料安全門偵測異常
      ANI     M1738  ; ROBOT緊急停止
      ANI     X30F  ; 進料ROBOT示教模式-OUT16
      ANI     M8010
      OUT     Y30F  ; 進料ROBOT外部停止(OFF停止)-IN16
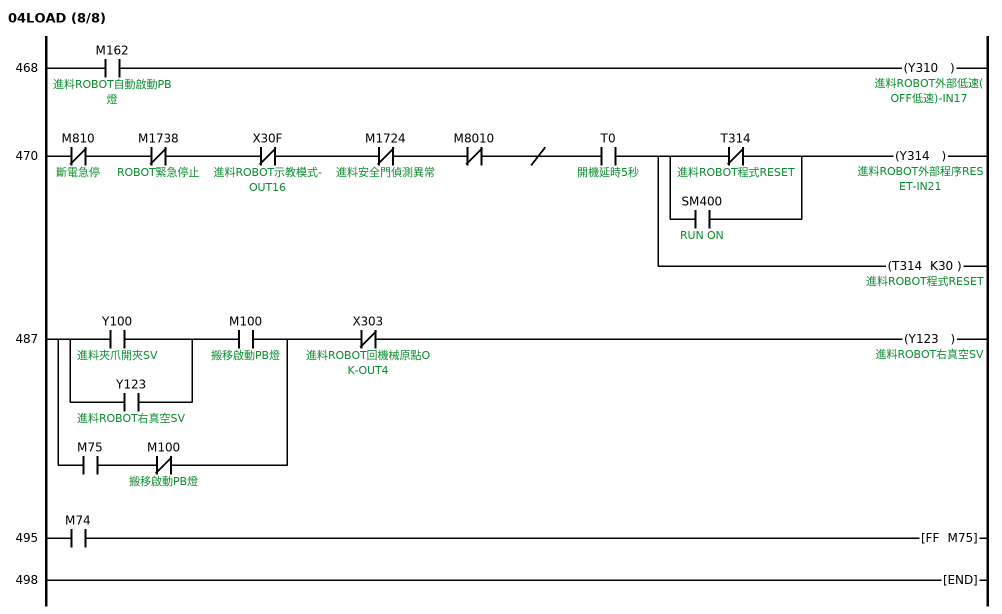
468   LD      M162  ; 進料ROBOT自動啟動PB燈
      OUT     Y310  ; 進料ROBOT外部低速(OFF低速)-IN17
470   LDI     M810  ; 斷電急停
      ANI     M1738  ; ROBOT緊急停止
      ANI     X30F  ; 進料ROBOT示教模式-OUT16
      ANI     M1724  ; 進料安全門偵測異常
      ANI     M8010
      INV
      AND     T0  ; 開機延時5秒
      MPS
      LDI     T314  ; 進料ROBOT程式RESET
      OR      SM400  ; RUN ON
      ANB
      OUT     Y314  ; 進料ROBOT外部程序RESET-IN21
      MPP
      OUT     T314 K30  ; 進料ROBOT程式RESET
487   LD      Y100  ; 進料夾爪開夾SV
      OR      Y123  ; 進料ROBOT右真空SV
      AND     M100  ; 搬移啟動PB燈
      LD      M75
      ANI     M100  ; 搬移啟動PB燈
      ORB
      ANI     X303  ; 進料ROBOT回機械原點OK-OUT4
      OUT     Y123  ; 進料ROBOT右真空SV
495   LD      M74
      FF      M75
498   END
END_PROGRAM

PROGRAM 05LOADUP
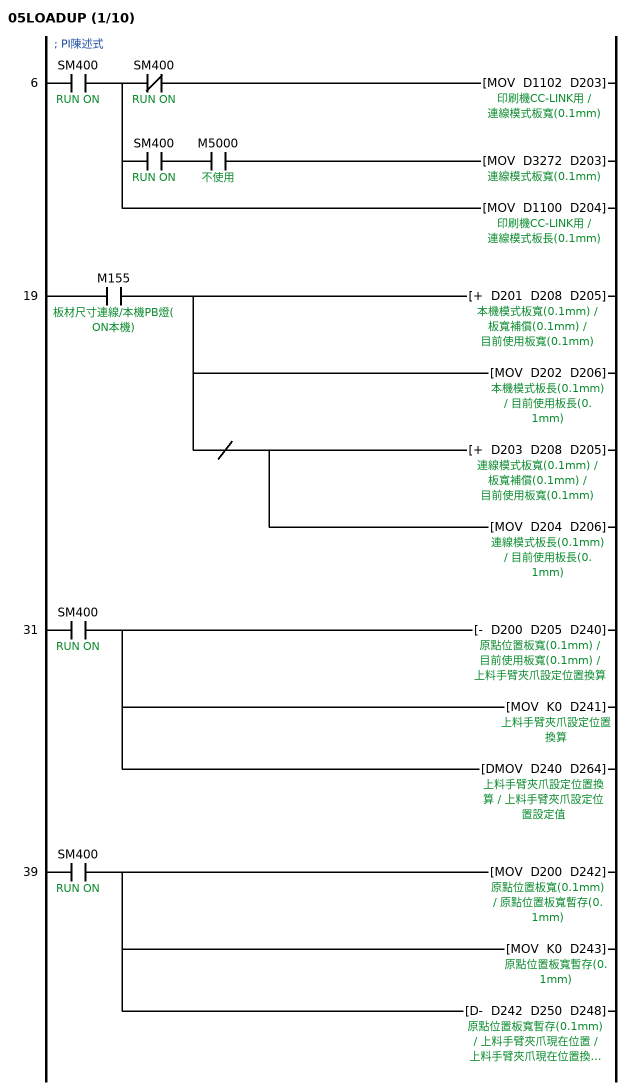
; PI陳述式
6     LD      SM400  ; RUN ON
      MPS
      ANI     SM400  ; RUN ON
      MOV     D1102 D203  ; 印刷機CC-LINK用 / 連線模式板寬(0.1mm)
      MRD
      AND     SM400  ; RUN ON
      AND     M5000  ; 不使用
      MOV     D3272 D203
      MPP
      MOV     D1100 D204  ; 印刷機CC-LINK用 / 連線模式板長(0.1mm)
19    LD      M155  ; 板材尺寸連線/本機PB燈(ON本機)
      +       D201 D208 D205  ; 本機模式板寬(0.1mm) / 板寬補償(0.1mm) / 目前使用板寬(0.1mm)
      MOV     D202 D206  ; 本機模式板長(0.1mm) / 目前使用板長(0.1mm)
      INV
      +       D203 D208 D205
      MOV     D204 D206
31    LD      SM400  ; RUN ON
      -       D200 D205 D240  ; 原點位置板寬(0.1mm) / 上料手臂夾爪設定位置換算
      MOV     K0 D241  ; 上料手臂夾爪設定位置換算
      DMOV    D240 D264  ; 上料手臂夾爪設定位置設定值
39    LD      SM400  ; RUN ON
      MOV     D200 D242  ; 原點位置板寬暫存(0.1mm)
      MOV     K0 D243  ; 原點位置板寬暫存(0.1mm)
      D-      D242 D250 D248  ; 上料手臂夾爪現在位置 / 上料手臂夾爪現在位置換算板寬
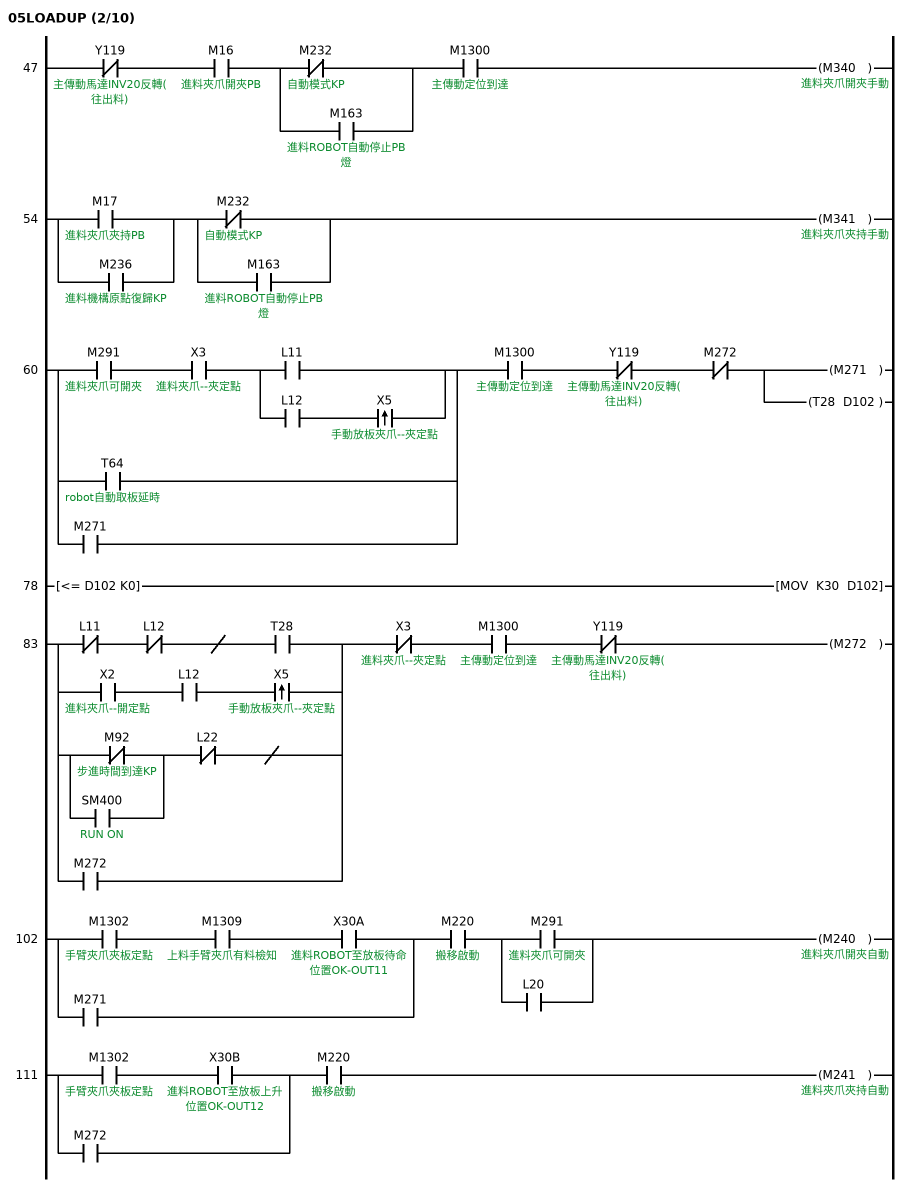
47    LDI     Y119  ; 主傳動馬達INV20反轉(往出料)
      AND     M16  ; 進料夾爪開夾PB
      LDI     M232  ; 自動模式KP
      OR      M163  ; 進料ROBOT自動停止PB燈
      ANB
      AND     M1300  ; 主傳動定位到達
      OUT     M340  ; 進料夾爪開夾手動
54    LD      M17  ; 進料夾爪夾持PB
      OR      M236  ; 進料機構原點復歸KP
      LDI     M232  ; 自動模式KP
      OR      M163  ; 進料ROBOT自動停止PB燈
      ANB
      OUT     M341  ; 進料夾爪夾持手動
60    LD      M291  ; 進料夾爪可開夾
      AND     X3  ; 進料夾爪--夾定點
      LD      L11
      LD      L12
      ANDP    X5  ; 手動放板夾爪--夾定點
      ORB
      ANB
      OR      T64  ; robot自動取板延時
      OR      M271
      AND     M1300  ; 主傳動定位到達
      ANI     Y119  ; 主傳動馬達INV20反轉(往出料)
      ANI     M272
      OUT     M271
      OUT     T28 D102
78    LD<=    D102 K0
      MOV     K30 D102
83    LDI     L11
      ANI     L12
      INV
      AND     T28
      LD      X2  ; 進料夾爪--開定點
      AND     L12
      ANDP    X5  ; 手動放板夾爪--夾定點
      ORB
      LDI     M92  ; 步進時間到達KP
      OR      SM400  ; RUN ON
      ANI     L22
      INV
      ORB
      OR      M272
      ANI     X3  ; 進料夾爪--夾定點
      AND     M1300  ; 主傳動定位到達
      ANI     Y119  ; 主傳動馬達INV20反轉(往出料)
      OUT     M272
102   LD      M1302  ; 手臂夾爪夾板定點
      AND     M1309  ; 上料手臂夾爪有料檢知
      AND     X30A  ; 進料ROBOT至放板待命位置OK-OUT11
      OR      M271
      AND     M220  ; 搬移啟動
      LD      M291  ; 進料夾爪可開夾
      OR      L20
      ANB
      OUT     M240  ; 進料夾爪開夾自動
111   LD      M1302  ; 手臂夾爪夾板定點
      AND     X30B  ; 進料ROBOT至放板上升位置OK-OUT12
      OR      M272
      AND     M220  ; 搬移啟動
      OUT     M241  ; 進料夾爪夾持自動
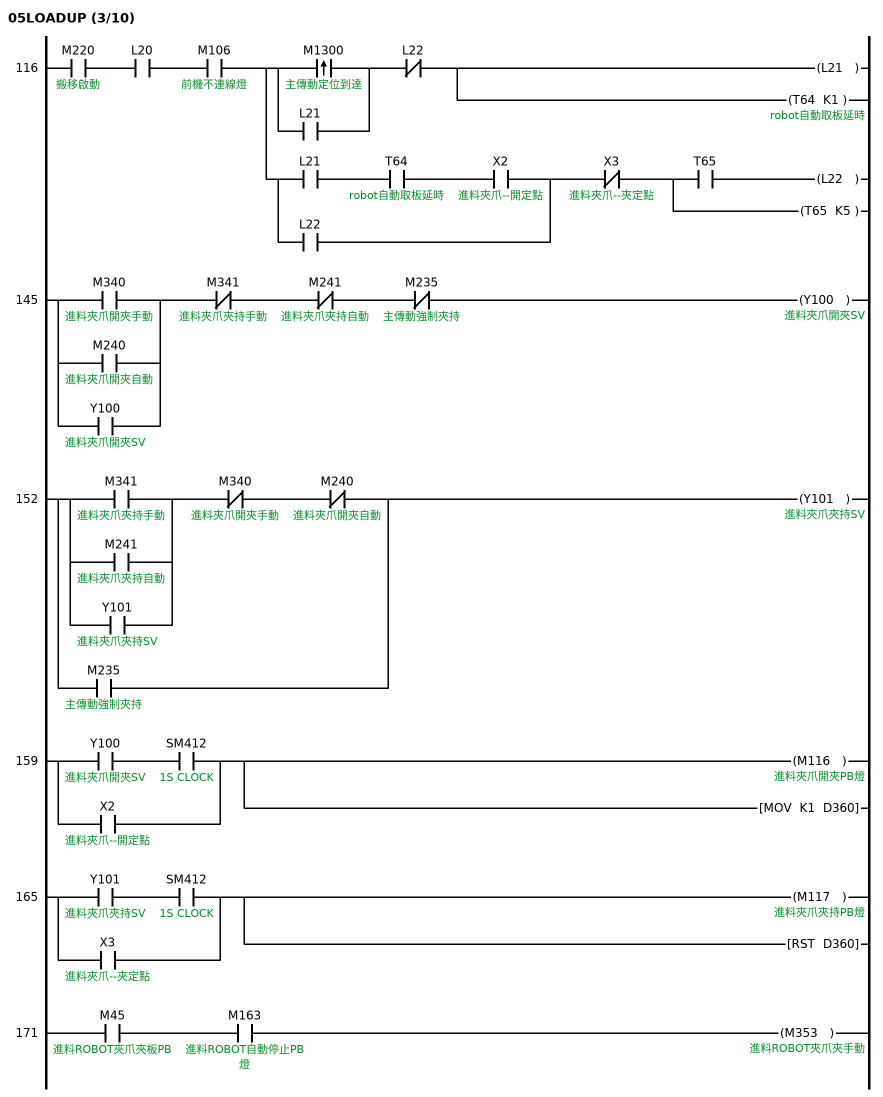
116   LD      M220  ; 搬移啟動
      AND     L20
      AND     M106  ; 前機不連線燈
      MPS
      LDP     M1300  ; 主傳動定位到達
      OR      L21
      ANB
      ANI     L22
      OUT     L21
      OUT     T64 K1  ; robot自動取板延時
      MPP
      LD      L21
      AND     T64  ; robot自動取板延時
      AND     X2  ; 進料夾爪--開定點
      OR      L22
      ANB
      ANI     X3  ; 進料夾爪--夾定點
      MPS
      AND     T65
      OUT     L22
      MPP
      OUT     T65 K5
145   LD      M340  ; 進料夾爪開夾手動
      OR      M240  ; 進料夾爪開夾自動
      OR      Y100  ; 進料夾爪開夾SV
      ANI     M341  ; 進料夾爪夾持手動
      ANI     M241  ; 進料夾爪夾持自動
      ANI     M235  ; 主傳動強制夾持
      OUT     Y100  ; 進料夾爪開夾SV
152   LD      M341  ; 進料夾爪夾持手動
      OR      M241  ; 進料夾爪夾持自動
      OR      Y101  ; 進料夾爪夾持SV
      ANI     M340  ; 進料夾爪開夾手動
      ANI     M240  ; 進料夾爪開夾自動
      OR      M235  ; 主傳動強制夾持
      OUT     Y101  ; 進料夾爪夾持SV
159   LD      Y100  ; 進料夾爪開夾SV
      AND     SM412  ; 1S CLOCK
      OR      X2  ; 進料夾爪--開定點
      OUT     M116  ; 進料夾爪開夾PB燈
      MOV     K1 D360
165   LD      Y101  ; 進料夾爪夾持SV
      AND     SM412  ; 1S CLOCK
      OR      X3  ; 進料夾爪--夾定點
      OUT     M117  ; 進料夾爪夾持PB燈
      RST     D360
171   LD      M45  ; 進料ROBOT夾爪夾板PB
      AND     M163  ; 進料ROBOT自動停止PB燈
      OUT     M353  ; 進料ROBOT夾爪夾手動
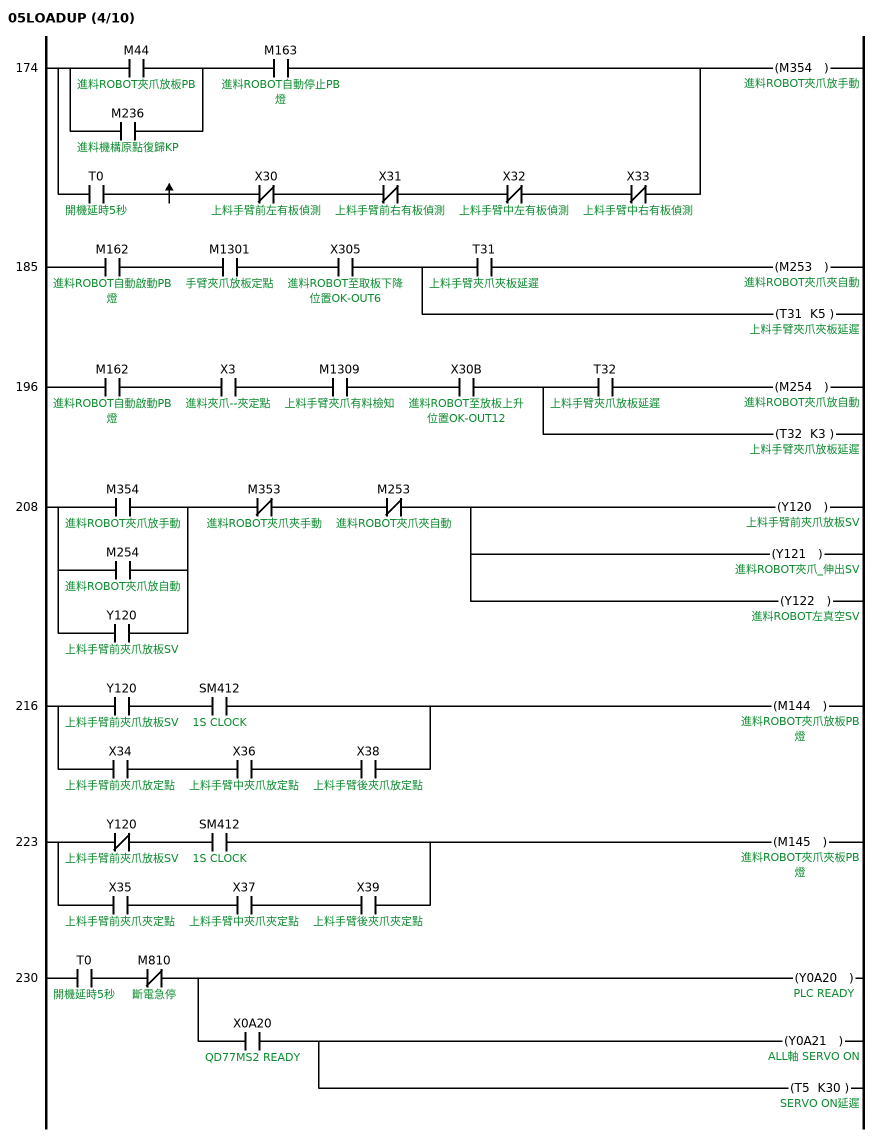
174   LD      M44  ; 進料ROBOT夾爪放板PB
      OR      M236  ; 進料機構原點復歸KP
      AND     M163  ; 進料ROBOT自動停止PB燈
      LD      T0  ; 開機延時5秒
      MEP
      ANI     X30  ; 上料手臂前左有板偵測
      ANI     X31  ; 上料手臂前右有板偵測
      ANI     X32  ; 上料手臂中左有板偵測
      ANI     X33  ; 上料手臂中右有板偵測
      ORB
      OUT     M354  ; 進料ROBOT夾爪放手動
185   LD      M162  ; 進料ROBOT自動啟動PB燈
      AND     M1301  ; 手臂夾爪放板定點
      AND     X305  ; 進料ROBOT至取板下降位置OK-OUT6
      MPS
      AND     T31  ; 上料手臂夾爪夾板延遲
      OUT     M253  ; 進料ROBOT夾爪夾自動
      MPP
      OUT     T31 K5  ; 上料手臂夾爪夾板延遲
196   LD      M162  ; 進料ROBOT自動啟動PB燈
      AND     X3  ; 進料夾爪--夾定點
      AND     M1309  ; 上料手臂夾爪有料檢知
      AND     X30B  ; 進料ROBOT至放板上升位置OK-OUT12
      MPS
      AND     T32  ; 上料手臂夾爪放板延遲
      OUT     M254  ; 進料ROBOT夾爪放自動
      MPP
      OUT     T32 K3  ; 上料手臂夾爪放板延遲
208   LD      M354  ; 進料ROBOT夾爪放手動
      OR      M254  ; 進料ROBOT夾爪放自動
      OR      Y120  ; 上料手臂前夾爪放板SV
      ANI     M353  ; 進料ROBOT夾爪夾手動
      ANI     M253  ; 進料ROBOT夾爪夾自動
      OUT     Y120  ; 上料手臂前夾爪放板SV
      OUT     Y121  ; 進料ROBOT夾爪_伸出SV
      OUT     Y122  ; 進料ROBOT左真空SV
216   LD      Y120  ; 上料手臂前夾爪放板SV
      AND     SM412  ; 1S CLOCK
      LD      X34  ; 上料手臂前夾爪放定點
      AND     X36  ; 上料手臂中夾爪放定點
      AND     X38  ; 上料手臂後夾爪放定點
      ORB
      OUT     M144  ; 進料ROBOT夾爪放板PB燈
223   LDI     Y120  ; 上料手臂前夾爪放板SV
      AND     SM412  ; 1S CLOCK
      LD      X35  ; 上料手臂前夾爪夾定點
      AND     X37  ; 上料手臂中夾爪夾定點
      AND     X39  ; 上料手臂後夾爪夾定點
      ORB
      OUT     M145  ; 進料ROBOT夾爪夾板PB燈
230   LD      T0  ; 開機延時5秒
      ANI     M810  ; 斷電急停
      OUT     Y0A20  ; PLC READY
      AND     X0A20  ; QD77MS2 READY
      OUT     Y0A21  ; ALL軸 SERVO ON
      OUT     T5 K30  ; SERVO ON延遲
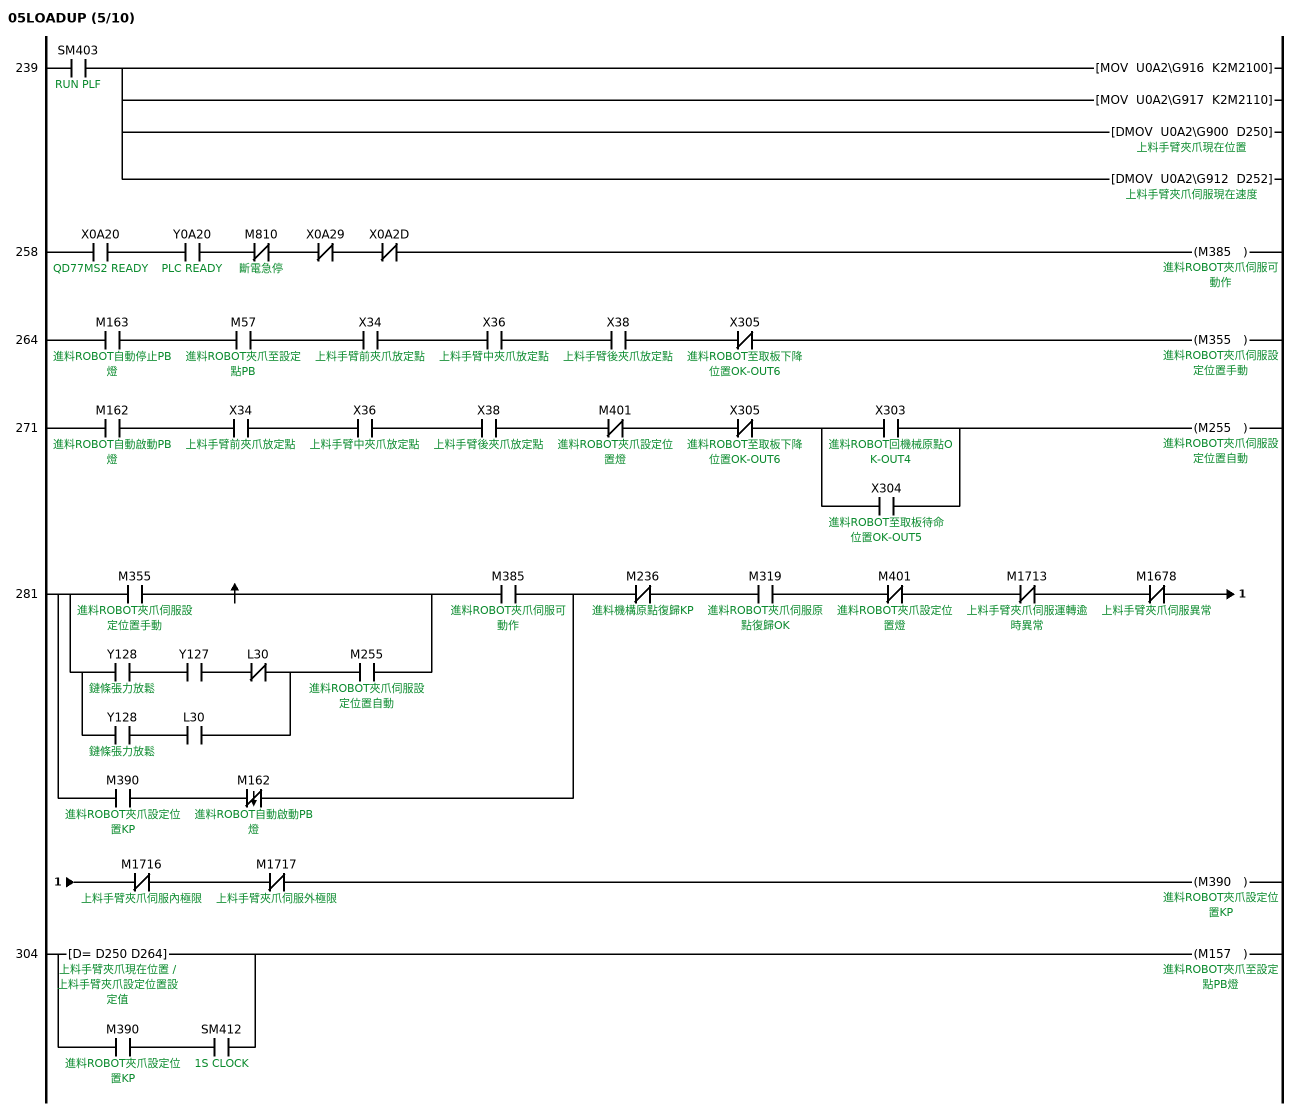
239   LD      SM403  ; RUN PLF
      MOV     U0A2\G916 K2M2100
      MOV     U0A2\G917 K2M2110
      DMOV    U0A2\G900 D250
      DMOV    U0A2\G912 D252  ; 上料手臂夾爪伺服現在速度
258   LD      X0A20  ; QD77MS2 READY
      AND     Y0A20  ; PLC READY
      ANI     M810  ; 斷電急停
      ANI     X0A29
      ANI     X0A2D
      OUT     M385  ; 進料ROBOT夾爪伺服可動作
264   LD      M163  ; 進料ROBOT自動停止PB燈
      AND     M57  ; 進料ROBOT夾爪至設定點PB
      AND     X34  ; 上料手臂前夾爪放定點
      AND     X36  ; 上料手臂中夾爪放定點
      AND     X38  ; 上料手臂後夾爪放定點
      ANI     X305  ; 進料ROBOT至取板下降位置OK-OUT6
      OUT     M355  ; 進料ROBOT夾爪伺服設定位置手動
271   LD      M162  ; 進料ROBOT自動啟動PB燈
      AND     X34  ; 上料手臂前夾爪放定點
      AND     X36  ; 上料手臂中夾爪放定點
      AND     X38  ; 上料手臂後夾爪放定點
      ANI     M401  ; 進料ROBOT夾爪設定位置燈
      ANI     X305  ; 進料ROBOT至取板下降位置OK-OUT6
      LD      X303  ; 進料ROBOT回機械原點OK-OUT4
      OR      X304  ; 進料ROBOT至取板待命位置OK-OUT5
      ANB
      OUT     M255  ; 進料ROBOT夾爪伺服設定位置自動
281   LD      M355  ; 進料ROBOT夾爪伺服設定位置手動
      MEP
      LD      Y128  ; 鏈條張力放鬆
      AND     Y127
      ANI     L30
      LD      Y128  ; 鏈條張力放鬆
      AND     L30
      ORB
      AND     M255  ; 進料ROBOT夾爪伺服設定位置自動
      ORB
      AND     M385  ; 進料ROBOT夾爪伺服可動作
      LD      M390  ; 進料ROBOT夾爪設定位置KP
      ANDFI   M162  ; 進料ROBOT自動啟動PB燈
      ORB
      ANI     M236  ; 進料機構原點復歸KP
      AND     M319  ; 進料ROBOT夾爪伺服原點復歸OK
      ANI     M401  ; 進料ROBOT夾爪設定位置燈
      ANI     M1713  ; 上料手臂夾爪伺服運轉逾時異常
      ANI     M1678  ; 上料手臂夾爪伺服異常
      ANI     M1716  ; 上料手臂夾爪伺服內極限
      ANI     M1717  ; 上料手臂夾爪伺服外極限
      OUT     M390  ; 進料ROBOT夾爪設定位置KP
304   LDD=    D250 D264  ; 上料手臂夾爪現在位置 / 上料手臂夾爪設定位置設定值
      LD      M390  ; 進料ROBOT夾爪設定位置KP
      AND     SM412  ; 1S CLOCK
      ORB
      OUT     M157  ; 進料ROBOT夾爪至設定點PB燈
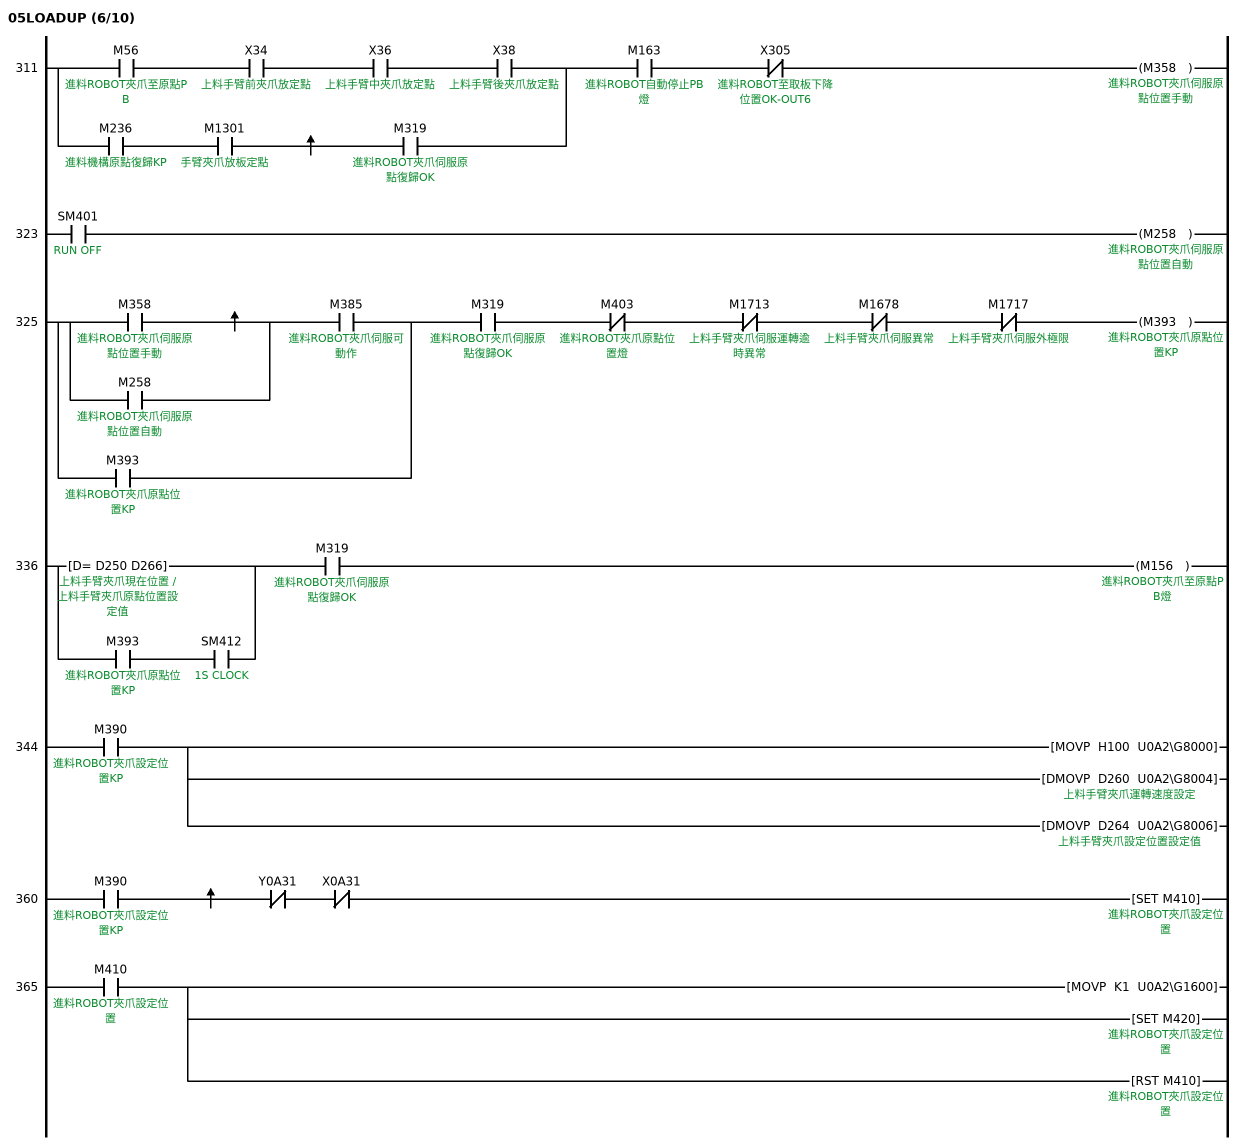
311   LD      M56  ; 進料ROBOT夾爪至原點PB
      AND     X34  ; 上料手臂前夾爪放定點
      AND     X36  ; 上料手臂中夾爪放定點
      AND     X38  ; 上料手臂後夾爪放定點
      LD      M236  ; 進料機構原點復歸KP
      AND     M1301  ; 手臂夾爪放板定點
      MEP
      AND     M319  ; 進料ROBOT夾爪伺服原點復歸OK
      ORB
      AND     M163  ; 進料ROBOT自動停止PB燈
      ANI     X305  ; 進料ROBOT至取板下降位置OK-OUT6
      OUT     M358  ; 進料ROBOT夾爪伺服原點位置手動
323   LD      SM401  ; RUN OFF
      OUT     M258  ; 進料ROBOT夾爪伺服原點位置自動
325   LD      M358  ; 進料ROBOT夾爪伺服原點位置手動
      MEP
      OR      M258  ; 進料ROBOT夾爪伺服原點位置自動
      AND     M385  ; 進料ROBOT夾爪伺服可動作
      OR      M393  ; 進料ROBOT夾爪原點位置KP
      AND     M319  ; 進料ROBOT夾爪伺服原點復歸OK
      ANI     M403  ; 進料ROBOT夾爪原點位置燈
      ANI     M1713  ; 上料手臂夾爪伺服運轉逾時異常
      ANI     M1678  ; 上料手臂夾爪伺服異常
      ANI     M1717  ; 上料手臂夾爪伺服外極限
      OUT     M393  ; 進料ROBOT夾爪原點位置KP
336   LDD=    D250 D266  ; 上料手臂夾爪現在位置 / 上料手臂夾爪原點位置設定值
      LD      M393  ; 進料ROBOT夾爪原點位置KP
      AND     SM412  ; 1S CLOCK
      ORB
      AND     M319  ; 進料ROBOT夾爪伺服原點復歸OK
      OUT     M156  ; 進料ROBOT夾爪至原點PB燈
344   LD      M390  ; 進料ROBOT夾爪設定位置KP
      MOVP    H100 U0A2\G8000
      DMOVP   D260 U0A2\G8004  ; 上料手臂夾爪運轉速度設定
      DMOVP   D264 U0A2\G8006
360   LD      M390  ; 進料ROBOT夾爪設定位置KP
      MEP
      ANI     Y0A31
      ANI     X0A31
      SET     M410  ; 進料ROBOT夾爪設定位置
365   LD      M410  ; 進料ROBOT夾爪設定位置
      MOVP    K1 U0A2\G1600
      SET     M420  ; 進料ROBOT夾爪設定位置
      RST     M410  ; 進料ROBOT夾爪設定位置
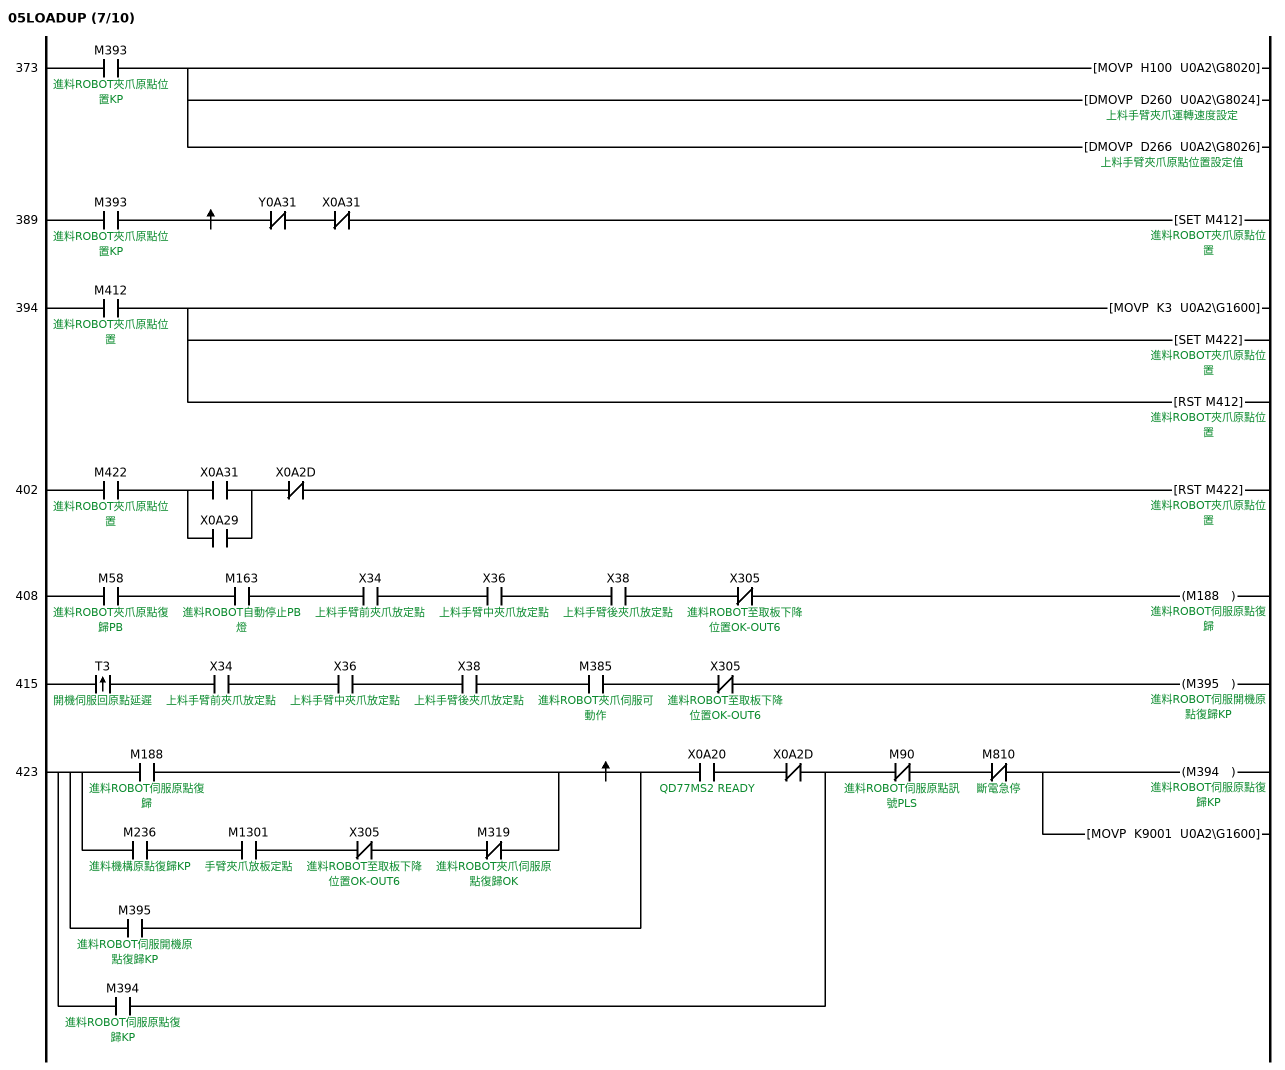
373   LD      M393  ; 進料ROBOT夾爪原點位置KP
      MOVP    H100 U0A2\G8020
      DMOVP   D260 U0A2\G8024
      DMOVP   D266 U0A2\G8026
389   LD      M393  ; 進料ROBOT夾爪原點位置KP
      MEP
      ANI     Y0A31
      ANI     X0A31
      SET     M412  ; 進料ROBOT夾爪原點位置
394   LD      M412  ; 進料ROBOT夾爪原點位置
      MOVP    K3 U0A2\G1600
      SET     M422  ; 進料ROBOT夾爪原點位置
      RST     M412  ; 進料ROBOT夾爪原點位置
402   LD      M422  ; 進料ROBOT夾爪原點位置
      LD      X0A31
      OR      X0A29
      ANB
      ANI     X0A2D
      RST     M422  ; 進料ROBOT夾爪原點位置
408   LD      M58  ; 進料ROBOT夾爪原點復歸PB
      AND     M163  ; 進料ROBOT自動停止PB燈
      AND     X34  ; 上料手臂前夾爪放定點
      AND     X36  ; 上料手臂中夾爪放定點
      AND     X38  ; 上料手臂後夾爪放定點
      ANI     X305  ; 進料ROBOT至取板下降位置OK-OUT6
      OUT     M188  ; 進料ROBOT伺服原點復歸
415   LDP     T3  ; 開機伺服回原點延遲
      AND     X34  ; 上料手臂前夾爪放定點
      AND     X36  ; 上料手臂中夾爪放定點
      AND     X38  ; 上料手臂後夾爪放定點
      AND     M385  ; 進料ROBOT夾爪伺服可動作
      ANI     X305  ; 進料ROBOT至取板下降位置OK-OUT6
      OUT     M395  ; 進料ROBOT伺服開機原點復歸KP
423   LD      M188  ; 進料ROBOT伺服原點復歸
      LD      M236  ; 進料機構原點復歸KP
      AND     M1301  ; 手臂夾爪放板定點
      ANI     X305  ; 進料ROBOT至取板下降位置OK-OUT6
      ANI     M319  ; 進料ROBOT夾爪伺服原點復歸OK
      ORB
      MEP
      OR      M395  ; 進料ROBOT伺服開機原點復歸KP
      AND     X0A20  ; QD77MS2 READY
      ANI     X0A2D
      OR      M394  ; 進料ROBOT伺服原點復歸KP
      ANI     M90  ; 進料ROBOT伺服原點訊號PLS
      ANI     M810  ; 斷電急停
      OUT     M394  ; 進料ROBOT伺服原點復歸KP
      MOVP    K9001 U0A2\G1600
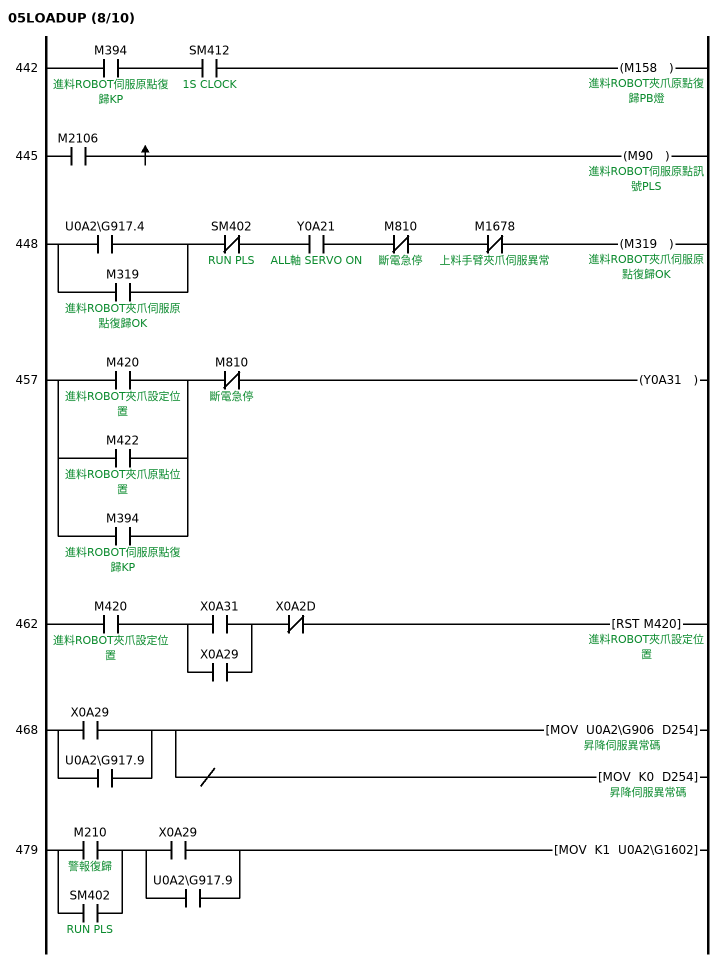
442   LD      M394  ; 進料ROBOT伺服原點復歸KP
      AND     SM412  ; 1S CLOCK
      OUT     M158  ; 進料ROBOT夾爪原點復歸PB燈
445   LD      M2106
      MEP
      OUT     M90  ; 進料ROBOT伺服原點訊號PLS
448   LD      U0A2\G917.4
      OR      M319  ; 進料ROBOT夾爪伺服原點復歸OK
      ANI     SM402  ; RUN PLS
      AND     Y0A21  ; ALL軸 SERVO ON
      ANI     M810  ; 斷電急停
      ANI     M1678  ; 上料手臂夾爪伺服異常
      OUT     M319  ; 進料ROBOT夾爪伺服原點復歸OK
457   LD      M420  ; 進料ROBOT夾爪設定位置
      OR      M422  ; 進料ROBOT夾爪原點位置
      OR      M394  ; 進料ROBOT伺服原點復歸KP
      ANI     M810  ; 斷電急停
      OUT     Y0A31
462   LD      M420  ; 進料ROBOT夾爪設定位置
      LD      X0A31
      OR      X0A29
      ANB
      ANI     X0A2D
      RST     M420  ; 進料ROBOT夾爪設定位置
468   LD      X0A29
      OR      U0A2\G917.9
      MOV     U0A2\G906 D254  ; 昇降伺服異常碼
      INV
      MOV     K0 D254
479   LD      M210  ; 警報復歸
      OR      SM402  ; RUN PLS
      LD      X0A29
      OR      U0A2\G917.9
      ANB
      MOV     K1 U0A2\G1602
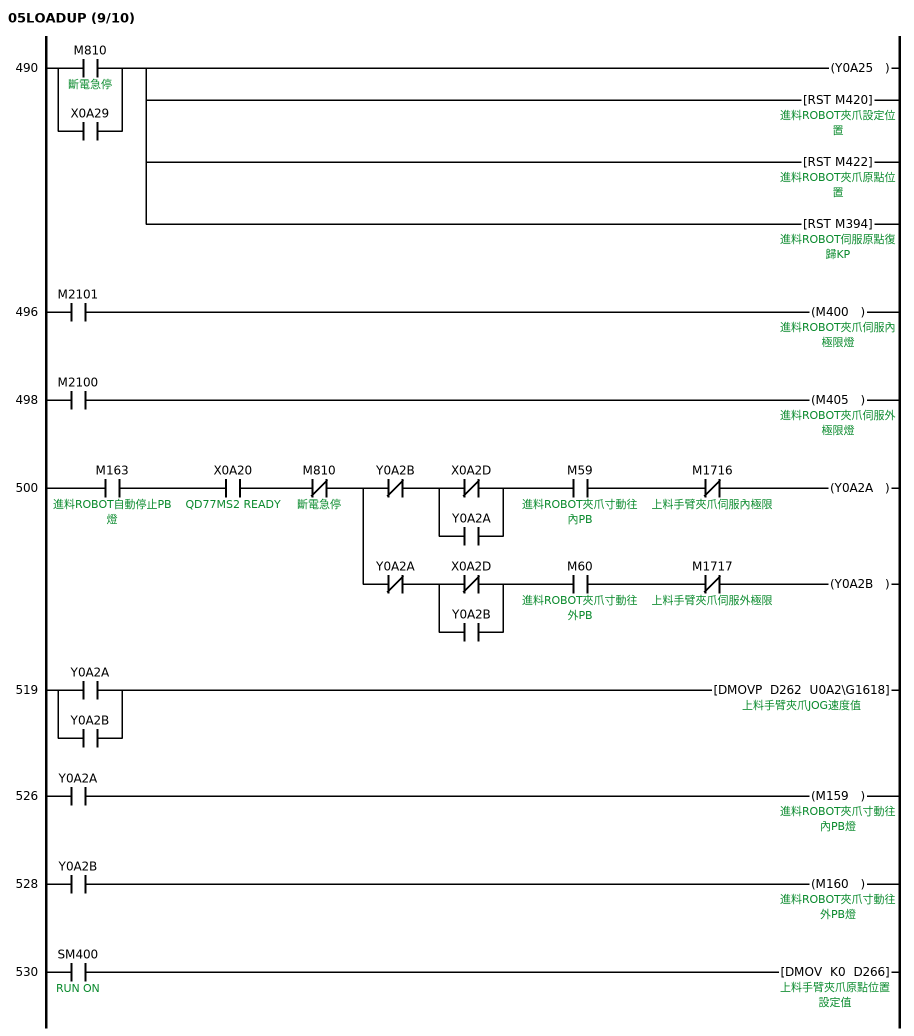
490   LD      M810  ; 斷電急停
      OR      X0A29
      OUT     Y0A25
      RST     M420  ; 進料ROBOT夾爪設定位置
      RST     M422  ; 進料ROBOT夾爪原點位置
      RST     M394  ; 進料ROBOT伺服原點復歸KP
496   LD      M2101
      OUT     M400  ; 進料ROBOT夾爪伺服內極限燈
498   LD      M2100
      OUT     M405  ; 進料ROBOT夾爪伺服外極限燈
500   LD      M163  ; 進料ROBOT自動停止PB燈
      AND     X0A20  ; QD77MS2 READY
      ANI     M810  ; 斷電急停
      MPS
      ANI     Y0A2B
      LDI     X0A2D
      OR      Y0A2A
      ANB
      AND     M59  ; 進料ROBOT夾爪寸動往內PB
      ANI     M1716  ; 上料手臂夾爪伺服內極限
      OUT     Y0A2A
      MPP
      ANI     Y0A2A
      LDI     X0A2D
      OR      Y0A2B
      ANB
      AND     M60  ; 進料ROBOT夾爪寸動往外PB
      ANI     M1717  ; 上料手臂夾爪伺服外極限
      OUT     Y0A2B
519   LD      Y0A2A
      OR      Y0A2B
      DMOVP   D262 U0A2\G1618  ; 上料手臂夾爪JOG速度值
526   LD      Y0A2A
      OUT     M159  ; 進料ROBOT夾爪寸動往內PB燈
528   LD      Y0A2B
      OUT     M160  ; 進料ROBOT夾爪寸動往外PB燈
530   LD      SM400  ; RUN ON
      DMOV    K0 D266
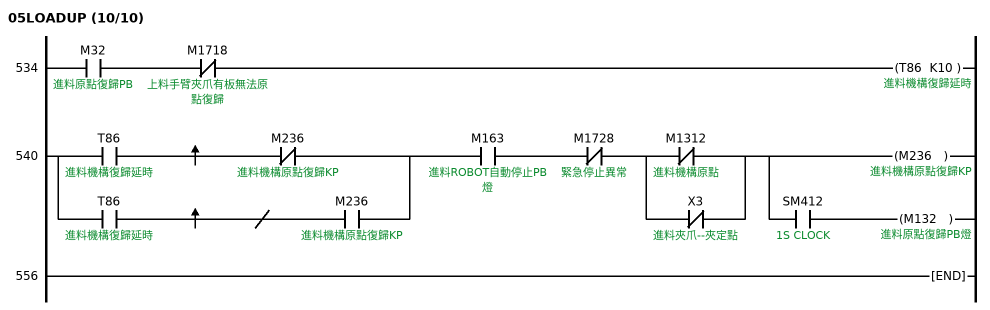
534   LD      M32  ; 進料原點復歸PB
      ANI     M1718  ; 上料手臂夾爪有板無法原點復歸
      OUT     T86 K10  ; 進料機構復歸延時
540   LD      T86  ; 進料機構復歸延時
      MEP
      ANI     M236  ; 進料機構原點復歸KP
      LD      T86  ; 進料機構復歸延時
      MEP
      INV
      AND     M236  ; 進料機構原點復歸KP
      ORB
      AND     M163  ; 進料ROBOT自動停止PB燈
      ANI     M1728  ; 緊急停止異常
      LDI     M1312  ; 進料機構原點
      ORI     X3  ; 進料夾爪--夾定點
      ANB
      OUT     M236  ; 進料機構原點復歸KP
      AND     SM412  ; 1S CLOCK
      OUT     M132  ; 進料原點復歸PB燈
556   END
END_PROGRAM

PROGRAM 06UNLOAD
